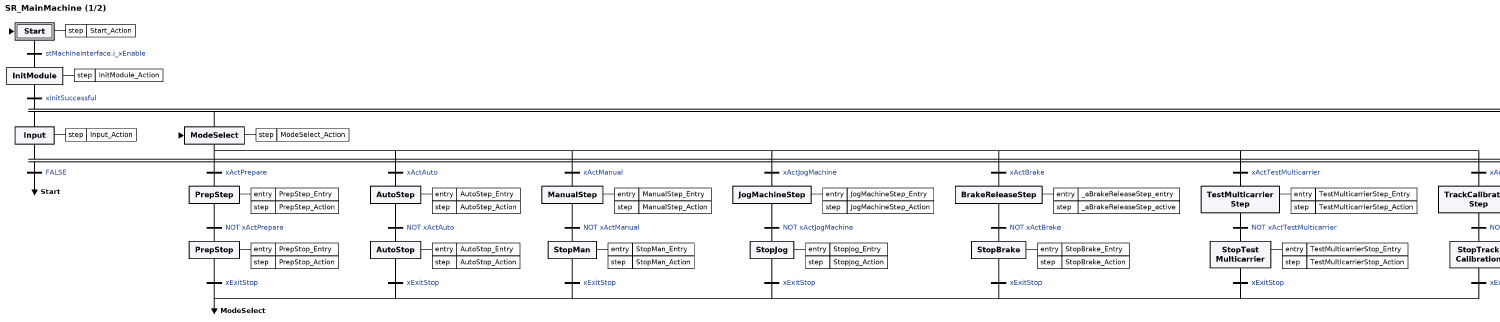
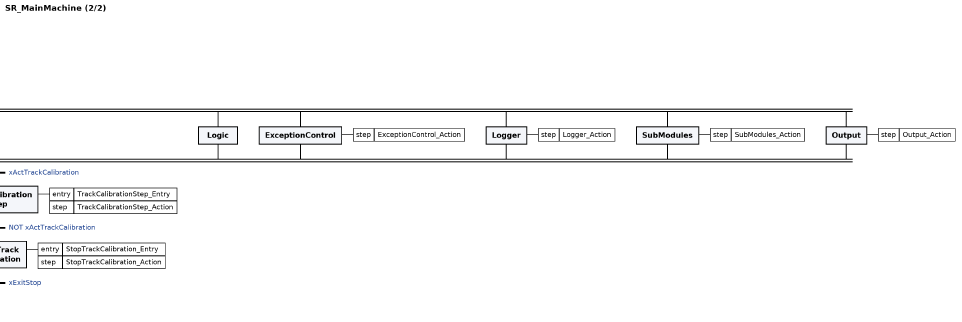
INITIAL_STEP Start:
    Start_Action(N);  // step action
END_STEP
TRANSITION FROM Start TO InitModule
    := stMachineInterface.i_xEnable;
END_TRANSITION
STEP InitModule:
    InitModule_Action(N);  // step action
END_STEP
TRANSITION FROM InitModule TO (Input, ModeSelect, Logic, ExceptionControl, Logger, SubModules, Output)
    := xInitSuccessful;
END_TRANSITION
STEP Input:
    Input_Action(N);  // step action
END_STEP
STEP ModeSelect:
    ModeSelect_Action(N);  // step action
END_STEP
TRANSITION FROM ModeSelect TO PrepStep
    := xActPrepare;
END_TRANSITION
STEP PrepStep:
    PrepStep_Entry(P1);  // entry action
    PrepStep_Action(N);  // step action
END_STEP
TRANSITION FROM PrepStep TO PrepStop
    := NOT xActPrepare;
END_TRANSITION
STEP PrepStop:
    PrepStop_Entry(P1);  // entry action
    PrepStop_Action(N);  // step action
END_STEP
TRANSITION FROM PrepStop TO ModeSelect
    := xExitStop;
END_TRANSITION
TRANSITION FROM ModeSelect TO AutoStep
    := xActAuto;
END_TRANSITION
STEP AutoStep:
    AutoStep_Entry(P1);  // entry action
    AutoStep_Action(N);  // step action
END_STEP
TRANSITION FROM AutoStep TO AutoStop
    := NOT xActAuto;
END_TRANSITION
STEP AutoStop:
    AutoStop_Entry(P1);  // entry action
    AutoStop_Action(N);  // step action
END_STEP
TRANSITION FROM AutoStop TO ModeSelect
    := xExitStop;
END_TRANSITION
TRANSITION FROM ModeSelect TO ManualStep
    := xActManual;
END_TRANSITION
STEP ManualStep:
    ManualStep_Entry(P1);  // entry action
    ManualStep_Action(N);  // step action
END_STEP
TRANSITION FROM ManualStep TO StopMan
    := NOT xActManual;
END_TRANSITION
STEP StopMan:
    StopMan_Entry(P1);  // entry action
    StopMan_Action(N);  // step action
END_STEP
TRANSITION FROM StopMan TO ModeSelect
    := xExitStop;
END_TRANSITION
TRANSITION FROM ModeSelect TO JogMachineStep
    := xActJogMachine;
END_TRANSITION
STEP JogMachineStep:
    JogMachineStep_Entry(P1);  // entry action
    JogMachineStep_Action(N);  // step action
END_STEP
TRANSITION FROM JogMachineStep TO StopJog
    := NOT xActJogMachine;
END_TRANSITION
STEP StopJog:
    StopJog_Entry(P1);  // entry action
    StopJog_Action(N);  // step action
END_STEP
TRANSITION FROM StopJog TO ModeSelect
    := xExitStop;
END_TRANSITION
TRANSITION FROM ModeSelect TO BrakeReleaseStep
    := xActBrake;
END_TRANSITION
STEP BrakeReleaseStep:
    _aBrakeReleaseStep_entry(P1);  // entry action
    _aBrakeReleaseStep_active(N);  // step action
END_STEP
TRANSITION FROM BrakeReleaseStep TO StopBrake
    := NOT xActBrake;
END_TRANSITION
STEP StopBrake:
    StopBrake_Entry(P1);  // entry action
    StopBrake_Action(N);  // step action
END_STEP
TRANSITION FROM StopBrake TO ModeSelect
    := xExitStop;
END_TRANSITION
TRANSITION FROM ModeSelect TO TestMulticarrierStep
    := xActTestMulticarrier;
END_TRANSITION
STEP TestMulticarrierStep:
    TestMulticarrierStep_Entry(P1);  // entry action
    TestMulticarrierStep_Action(N);  // step action
END_STEP
TRANSITION FROM TestMulticarrierStep TO StopTestMulticarrier
    := NOT xActTestMulticarrier;
END_TRANSITION
STEP StopTestMulticarrier:
    TestMulticarrierStop_Entry(P1);  // entry action
    TestMulticarrierStop_Action(N);  // step action
END_STEP
TRANSITION FROM StopTestMulticarrier TO ModeSelect
    := xExitStop;
END_TRANSITION
TRANSITION FROM ModeSelect TO TrackCalibrationStep
    := xActTrackCalibration;
END_TRANSITION
STEP TrackCalibrationStep:
    TrackCalibrationStep_Entry(P1);  // entry action
    TrackCalibrationStep_Action(N);  // step action
END_STEP
TRANSITION FROM TrackCalibrationStep TO StopTrackCalibration
    := NOT xActTrackCalibration;
END_TRANSITION
STEP StopTrackCalibration:
    StopTrackCalibration_Entry(P1);  // entry action
    StopTrackCalibration_Action(N);  // step action
END_STEP
TRANSITION FROM StopTrackCalibration TO ModeSelect
    := xExitStop;
END_TRANSITION
STEP Logic:
END_STEP
STEP ExceptionControl:
    ExceptionControl_Action(N);  // step action
END_STEP
STEP Logger:
    Logger_Action(N);  // step action
END_STEP
STEP SubModules:
    SubModules_Action(N);  // step action
END_STEP
STEP Output:
    Output_Action(N);  // step action
END_STEP
TRANSITION FROM (Input, Logic, ExceptionControl, Logger, SubModules, Output) TO Start
    := FALSE;
END_TRANSITION

ACTION Init_CmdTables:
(* System generated code, could be modified for your application *)

//-------------------------------------------------------------------------------------------------------------------
//-- Prepare  --
	//
	TPL.FC_FirstStep(udiStepIndex, diStep);
	astPrepareTable[udiStepIndex].sTitle					:= 'Prepare AllSubModules';
	astPrepareTable[udiStepIndex].udiModuleName				:= TPL.Gc_udiAllSubModules;
	astPrepareTable[udiStepIndex].diStep					:= diStep;
	astPrepareTable[udiStepIndex].diCMD						:= ET_Cmd.Prepare;
	astPrepareTable[udiStepIndex].timTimeOut				:= T#0MS;
	astPrepareTable[udiStepIndex].xEndCMD					:= FALSE;
	
	TPL.FC_LastStep(udiStepIndex, diStep);
	astPrepareTable[udiStepIndex].sTitle					:= 'End';
	astPrepareTable[udiStepIndex].udiModuleName				:= 0;
	astPrepareTable[udiStepIndex].diStep					:= diStep;
	astPrepareTable[udiStepIndex].diCMD						:= 0;
	astPrepareTable[udiStepIndex].timTimeOut				:= T#0MS;
	astPrepareTable[udiStepIndex].xEndCMD					:= TRUE;
	
	TPL.FC_FirstCmdTable(iq_udiTableIndex:= udiTableIndex);
	astListofCMDTables[udiTableIndex].diCMD					:= ET_Cmd.Prepare;
	astListofCMDTables[udiTableIndex].sTitle				:= 'Prepare';
	astListofCMDTables[udiTableIndex].udiNumberOfCmdSteps	:= udiStepIndex;

//-------------------------------------------------------------------------------------------------------------------
//-- StopPrepare  --
	//
	TPL.FC_FirstStep(udiStepIndex, diStep);
	astStopPrepareTable[udiStepIndex].sTitle					:= 'Stop Alpha + Bravo';
	astStopPrepareTable[udiStepIndex].udiModuleName				:= c_udiServoDrivesGroup;
	astStopPrepareTable[udiStepIndex].diStep					:= diStep;
	astStopPrepareTable[udiStepIndex].diCMD						:= ET_Cmd.Stop;
	astStopPrepareTable[udiStepIndex].timTimeOut				:= T#0MS;
	astStopPrepareTable[udiStepIndex].xEndCMD					:= FALSE;
	
	TPL.FC_NextStep(udiStepIndex, diStep);
	astStopPrepareTable[udiStepIndex].sTitle					:= 'Hold MultiCarrier';
	astStopPrepareTable[udiStepIndex].udiModuleName				:= c_udiMultiCarrier;
	astStopPrepareTable[udiStepIndex].diStep					:= diStep;
	astStopPrepareTable[udiStepIndex].diCMD						:= ET_Cmd.Hold;
	astStopPrepareTable[udiStepIndex].timTimeOut				:= T#0MS;
	astStopPrepareTable[udiStepIndex].xEndCMD					:= FALSE;
	
	TPL.FC_LastStep(udiStepIndex, diStep);
	astStopPrepareTable[udiStepIndex].sTitle					:= 'End';
	astStopPrepareTable[udiStepIndex].udiModuleName				:= 0;
	astStopPrepareTable[udiStepIndex].diStep					:= diStep;
	astStopPrepareTable[udiStepIndex].diCMD						:= 0;
	astStopPrepareTable[udiStepIndex].timTimeOut				:= T#0MS;
	astStopPrepareTable[udiStepIndex].xEndCMD					:= TRUE;
	
	TPL.FC_NextCmdTable(iq_udiTableIndex:= udiTableIndex);
	astListofCMDTables[udiTableIndex].diCMD						:= ET_Cmd.StopPrepare;
	astListofCMDTables[udiTableIndex].sTitle					:= 'StopPrepare';
	astListofCMDTables[udiTableIndex].udiNumberOfCmdSteps		:= udiStepIndex;
	
	
//-------------------------------------------------------------------------------------------------------------------
//-- Auto  --
	//
	TPL.FC_FirstStep(udiStepIndex, diStep);
	astAutoTable[udiStepIndex].sTitle						:= 'Auto Bravo';
	astAutoTable[udiStepIndex].udiModuleName				:= c_udiBravo;
	astAutoTable[udiStepIndex].diStep						:= diStep;
	astAutoTable[udiStepIndex].diCMD						:= ET_Cmd.Auto;
	astAutoTable[udiStepIndex].timTimeOut					:= T#0MS;
	astAutoTable[udiStepIndex].xEndCMD						:= FALSE;
	
	TPL.FC_NextStep(udiStepIndex, diStep);
	astAutoTable[udiStepIndex].sTitle						:= 'Auto Alpha';
	astAutoTable[udiStepIndex].udiModuleName				:= c_udiAlpha;
	astAutoTable[udiStepIndex].diStep						:= diStep;
	astAutoTable[udiStepIndex].diCMD						:= ET_Cmd.Auto;
	astAutoTable[udiStepIndex].timTimeOut					:= T#0MS;
	astAutoTable[udiStepIndex].xEndCMD						:= FALSE;
	
	TPL.FC_NextStep(udiStepIndex, diStep);
	astAutoTable[udiStepIndex].sTitle						:= 'Auto MultiCarrier';
	astAutoTable[udiStepIndex].udiModuleName				:= c_udiMultiCarrier;
	astAutoTable[udiStepIndex].diStep						:= diStep;
	astAutoTable[udiStepIndex].diCMD						:= ET_Cmd.Auto;
	astAutoTable[udiStepIndex].timTimeOut					:= T#0MS;
	astAutoTable[udiStepIndex].xEndCMD						:= FALSE;
	
	TPL.FC_LastStep(udiStepIndex, diStep);
	astAutoTable[udiStepIndex].sTitle						:= 'End';
	astAutoTable[udiStepIndex].udiModuleName				:= 0;
	astAutoTable[udiStepIndex].diStep						:= diStep;
	astAutoTable[udiStepIndex].diCMD						:= 0;
	astAutoTable[udiStepIndex].timTimeOut					:= T#0MS;
	astAutoTable[udiStepIndex].xEndCMD						:= TRUE;
	
	TPL.FC_NextCmdTable(iq_udiTableIndex:= udiTableIndex);
	astListofCMDTables[udiTableIndex].diCMD					:= ET_Cmd.Auto;
	astListofCMDTables[udiTableIndex].sTitle				:= 'Auto';
	astListofCMDTables[udiTableIndex].udiNumberOfCmdSteps	:= udiStepIndex;

//-------------------------------------------------------------------------------------------------------------------
//-- StopAuto --
	//
	TPL.FC_FirstStep(udiStepIndex, diStep);
	astStopAutoTable[udiStepIndex].sTitle					:= 'Hold Alpha';
	astStopAutoTable[udiStepIndex].udiModuleName			:= c_udiAlpha;
	astStopAutoTable[udiStepIndex].diStep					:= diStep;
	astStopAutoTable[udiStepIndex].diCMD					:= ET_Cmd.Hold;
	astStopAutoTable[udiStepIndex].timTimeOut				:= T#0MS;
	astStopAutoTable[udiStepIndex].xEndCMD					:= FALSE;
	
	TPL.FC_NextStep(udiStepIndex, diStep);
	astStopAutoTable[udiStepIndex].sTitle					:= 'Stop MultiCarrier';
	astStopAutoTable[udiStepIndex].udiModuleName			:= c_udiMultiCarrier;
	astStopAutoTable[udiStepIndex].diStep					:= diStep;
	astStopAutoTable[udiStepIndex].diCMD					:= ET_Cmd.Stop;
	astStopAutoTable[udiStepIndex].timTimeOut				:= T#0MS;
	astStopAutoTable[udiStepIndex].xEndCMD					:= FALSE;
	
	TPL.FC_LastStep(udiStepIndex, diStep);
	astStopAutoTable[udiStepIndex].sTitle					:= 'End';
	astStopAutoTable[udiStepIndex].udiModuleName			:= 0;
	astStopAutoTable[udiStepIndex].diStep					:= diStep;
	astStopAutoTable[udiStepIndex].diCMD					:= 0;
	astStopAutoTable[udiStepIndex].timTimeOut				:= T#0MS;
	astStopAutoTable[udiStepIndex].xEndCMD					:= TRUE;
	
	TPL.FC_NextCmdTable(iq_udiTableIndex:= udiTableIndex);
	astListofCMDTables[udiTableIndex].diCMD						:= ET_Cmd.StopAuto;
	astListofCMDTables[udiTableIndex].sTitle					:= 'StopAuto';
	astListofCMDTables[udiTableIndex].udiNumberOfCmdSteps		:= udiStepIndex;
	
	
	
//-------------------------------------------------------------------------------------------------------------------
//-- Manual  --
	//
	TPL.FC_FirstStep(udiStepIndex, diStep);
	astManualTable[udiStepIndex].sTitle						:= 'Stop AllSubModules';
	astManualTable[udiStepIndex].udiModuleName				:= TPL.Gc_udiAllSubModules;
	astManualTable[udiStepIndex].diStep						:= diStep;
	astManualTable[udiStepIndex].diCMD						:= ET_Cmd.Stop;
	astManualTable[udiStepIndex].timTimeOut					:= T#0MS;
	astManualTable[udiStepIndex].xEndCMD					:= FALSE;
	
	TPL.FC_NextStep(udiStepIndex, diStep);
	astManualTable[udiStepIndex].sTitle						:= 'Manual SlaveGroup';
	astManualTable[udiStepIndex].udiModuleName				:= TPL.Gc_udiAllSubModules;
	astManualTable[udiStepIndex].diStep						:= diStep;
	astManualTable[udiStepIndex].diCMD						:= ET_Cmd.Manual;
	astManualTable[udiStepIndex].timTimeOut					:= T#0MS;
	astManualTable[udiStepIndex].xEndCMD					:= FALSE;
	
	TPL.FC_LastStep(udiStepIndex, diStep);
	astManualTable[udiStepIndex].sTitle						:= 'End';
	astManualTable[udiStepIndex].udiModuleName				:= 0;
	astManualTable[udiStepIndex].diStep						:= diStep;
	astManualTable[udiStepIndex].diCMD						:= 0;
	astManualTable[udiStepIndex].timTimeOut					:= T#0MS;
	astManualTable[udiStepIndex].xEndCMD					:= TRUE;
	
	TPL.FC_NextCmdTable(iq_udiTableIndex:= udiTableIndex);
	astListofCMDTables[udiTableIndex].diCMD					:= ET_Cmd.Manual;
	astListofCMDTables[udiTableIndex].sTitle				:= 'Manual';
	astListofCMDTables[udiTableIndex].udiNumberOfCmdSteps	:= udiStepIndex;

//-------------------------------------------------------------------------------------------------------------------
//-- TestMulticarrier --
	//
	TPL.FC_FirstStep(udiStepIndex, diStep);
	astTestMulticarrierTable[udiStepIndex].sTitle						:= 'TestMulticarrier';
	astTestMulticarrierTable[udiStepIndex].udiModuleName				:= c_udiMultiCarrier;
	astTestMulticarrierTable[udiStepIndex].diStep						:= diStep;
	astTestMulticarrierTable[udiStepIndex].diCMD						:= ET_Cmd.TestMulticarrier;
	astTestMulticarrierTable[udiStepIndex].timTimeOut					:= T#0MS;
	astTestMulticarrierTable[udiStepIndex].xEndCMD						:= FALSE;
	
	TPL.FC_LastStep(udiStepIndex, diStep);
	astTestMulticarrierTable[udiStepIndex].sTitle						:= 'End';
	astTestMulticarrierTable[udiStepIndex].udiModuleName				:= 0;
	astTestMulticarrierTable[udiStepIndex].diStep						:= diStep;
	astTestMulticarrierTable[udiStepIndex].diCMD						:= 0;
	astTestMulticarrierTable[udiStepIndex].timTimeOut					:= T#0MS;
	astTestMulticarrierTable[udiStepIndex].xEndCMD						:= TRUE;
	
	TPL.FC_NextCmdTable(iq_udiTableIndex:= udiTableIndex);
	astListofCMDTables[udiTableIndex].diCMD					:= ET_Cmd.TestMulticarrier;
	astListofCMDTables[udiTableIndex].sTitle				:= 'TestMulticarrier';
	astListofCMDTables[udiTableIndex].udiNumberOfCmdSteps	:= udiStepIndex;
	
//-------------------------------------------------------------------------------------------------------------------
//-- TrackCalibration --
	//
	TPL.FC_FirstStep(udiStepIndex, diStep);
	astTrackCalibrationTable[udiStepIndex].sTitle						:= 'TrackCalibration';
	astTrackCalibrationTable[udiStepIndex].udiModuleName				:= c_udiMultiCarrier;
	astTrackCalibrationTable[udiStepIndex].diStep						:= diStep;
	astTrackCalibrationTable[udiStepIndex].diCMD						:= ET_Cmd.TrackCalibration;
	astTrackCalibrationTable[udiStepIndex].timTimeOut					:= T#0MS;
	astTrackCalibrationTable[udiStepIndex].xEndCMD						:= FALSE;
	
	TPL.FC_LastStep(udiStepIndex, diStep);
	astTrackCalibrationTable[udiStepIndex].sTitle						:= 'End';
	astTrackCalibrationTable[udiStepIndex].udiModuleName				:= 0;
	astTrackCalibrationTable[udiStepIndex].diStep						:= diStep;
	astTrackCalibrationTable[udiStepIndex].diCMD						:= 0;
	astTrackCalibrationTable[udiStepIndex].timTimeOut					:= T#0MS;
	astTrackCalibrationTable[udiStepIndex].xEndCMD						:= TRUE;
	
	TPL.FC_NextCmdTable(iq_udiTableIndex:= udiTableIndex);
	astListofCMDTables[udiTableIndex].diCMD					:= ET_Cmd.TrackCalibration;
	astListofCMDTables[udiTableIndex].sTitle				:= 'TrackCalibration';
	astListofCMDTables[udiTableIndex].udiNumberOfCmdSteps	:= udiStepIndex;
	
//-------------------------------------------------------------------------------------------------------------------
//-- Stop --
	//
	TPL.FC_FirstStep(udiStepIndex, diStep);
	astStopTable[udiStepIndex].sTitle						:= 'Stop AllSubModules';
	astStopTable[udiStepIndex].udiModuleName				:= TPL.Gc_udiAllSubModules;
	astStopTable[udiStepIndex].diStep						:= diStep;
	astStopTable[udiStepIndex].diCMD						:= ET_Cmd.Stop;
	astStopTable[udiStepIndex].timTimeOut					:= T#0MS;
	astStopTable[udiStepIndex].xEndCMD						:= FALSE;
	
	TPL.FC_LastStep(udiStepIndex, diStep);
	astStopTable[udiStepIndex].sTitle						:= 'End';
	astStopTable[udiStepIndex].udiModuleName				:= 0;
	astStopTable[udiStepIndex].diStep						:= diStep;
	astStopTable[udiStepIndex].diCMD						:= 0;
	astStopTable[udiStepIndex].timTimeOut					:= T#0MS;
	astStopTable[udiStepIndex].xEndCMD						:= TRUE;
	
	TPL.FC_NextCmdTable(iq_udiTableIndex:= udiTableIndex);
	astListofCMDTables[udiTableIndex].diCMD					:= ET_Cmd.Stop;
	astListofCMDTables[udiTableIndex].sTitle				:= 'Stop';
	astListofCMDTables[udiTableIndex].udiNumberOfCmdSteps	:= udiStepIndex;

//-------------------------------------------------------------------------------------------------------------------
//-- Start --
	//
	TPL.FC_FirstStep(udiStepIndex, diStep);
	astStartTable[udiStepIndex].sTitle						:= 'Start AllSubModules';
	astStartTable[udiStepIndex].udiModuleName				:= TPL.Gc_udiAllSubModules;
	astStartTable[udiStepIndex].diStep						:= diStep;
	astStartTable[udiStepIndex].diCMD						:= ET_Cmd.Start;
	astStartTable[udiStepIndex].timTimeOut					:= T#0MS;
	astStartTable[udiStepIndex].xEndCMD						:= FALSE;
	
	TPL.FC_LastStep(udiStepIndex, diStep);
	astStartTable[udiStepIndex].sTitle						:= 'End';
	astStartTable[udiStepIndex].udiModuleName				:= 0;
	astStartTable[udiStepIndex].diStep						:= diStep;
	astStartTable[udiStepIndex].diCMD						:= 0;
	astStartTable[udiStepIndex].timTimeOut					:= T#0MS;
	astStartTable[udiStepIndex].xEndCMD						:= TRUE;
	
	TPL.FC_NextCmdTable(iq_udiTableIndex:= udiTableIndex);
	astListofCMDTables[udiTableIndex].diCMD					:= ET_Cmd.Start;
	astListofCMDTables[udiTableIndex].sTitle				:= 'Start';
	astListofCMDTables[udiTableIndex].udiNumberOfCmdSteps	:= udiStepIndex;
	
//-------------------------------------------------------------------------------------------------------------------
//-- Abort --
	//
	TPL.FC_FirstStep(udiStepIndex, diStep);
	astAbortTable[udiStepIndex].sTitle						:= 'Abort AllSubModules';
	astAbortTable[udiStepIndex].udiModuleName				:= TPL.Gc_udiAllSubModules;
	astAbortTable[udiStepIndex].diStep						:= diStep;
	astAbortTable[udiStepIndex].diCMD						:= ET_Cmd.Abort;
	astAbortTable[udiStepIndex].timTimeOut					:= T#0MS;
	astAbortTable[udiStepIndex].xEndCMD						:= FALSE;
	
	TPL.FC_LastStep(udiStepIndex, diStep);
	astAbortTable[udiStepIndex].sTitle						:= 'End';
	astAbortTable[udiStepIndex].udiModuleName				:= 0;
	astAbortTable[udiStepIndex].diStep						:= diStep;
	astAbortTable[udiStepIndex].diCMD						:= 0;
	astAbortTable[udiStepIndex].timTimeOut					:= T#0MS;
	astAbortTable[udiStepIndex].xEndCMD						:= TRUE;
	
	TPL.FC_NextCmdTable(iq_udiTableIndex:= udiTableIndex);
	astListofCMDTables[udiTableIndex].diCMD					:= ET_Cmd.Abort;
	astListofCMDTables[udiTableIndex].sTitle				:= 'Abort';
	astListofCMDTables[udiTableIndex].udiNumberOfCmdSteps	:= udiStepIndex;

//-------------------------------------------------------------------------------------------------------------------
//-- Hold --
	//
	TPL.FC_FirstStep(udiStepIndex, diStep);
	astHoldTable[udiStepIndex].sTitle						:= 'Hold Alpha';
	astHoldTable[udiStepIndex].udiModuleName				:= c_udiAlpha;
	astHoldTable[udiStepIndex].diStep						:= diStep;
	astHoldTable[udiStepIndex].diCMD						:= ET_Cmd.Hold;
	astHoldTable[udiStepIndex].timTimeOut					:= T#0MS;
	astHoldTable[udiStepIndex].xEndCMD						:= FALSE;
	
	TPL.FC_LastStep(udiStepIndex, diStep);
	astHoldTable[udiStepIndex].sTitle						:= 'End';
	astHoldTable[udiStepIndex].udiModuleName				:= 0;
	astHoldTable[udiStepIndex].diStep						:= diStep;
	astHoldTable[udiStepIndex].diCMD						:= 0;
	astHoldTable[udiStepIndex].timTimeOut					:= T#0MS;
	astHoldTable[udiStepIndex].xEndCMD						:= TRUE;
	
	TPL.FC_NextCmdTable(iq_udiTableIndex:= udiTableIndex);
	astListofCMDTables[udiTableIndex].diCMD					:= ET_Cmd.Hold;
	astListofCMDTables[udiTableIndex].sTitle				:= 'Hold';
	astListofCMDTables[udiTableIndex].udiNumberOfCmdSteps	:= udiStepIndex;

//-------------------------------------------------------------------------------------------------------------------
//-- Hold for JogMachine --
	//
	TPL.FC_FirstStep(udiStepIndex, diStep);
	astHoldJogMachineTable[udiStepIndex].sTitle				:= 'Stop Alpha';
	astHoldJogMachineTable[udiStepIndex].udiModuleName		:= c_udiAlpha;
	astHoldJogMachineTable[udiStepIndex].diStep				:= diStep;
	astHoldJogMachineTable[udiStepIndex].diCMD				:= ET_Cmd.Stop;
	astHoldJogMachineTable[udiStepIndex].timTimeOut			:= T#0MS;
	astHoldJogMachineTable[udiStepIndex].xEndCMD			:= FALSE;
	
	TPL.FC_LastStep(udiStepIndex, diStep);
	astHoldJogMachineTable[udiStepIndex].sTitle				:= 'End';
	astHoldJogMachineTable[udiStepIndex].udiModuleName		:= 0;
	astHoldJogMachineTable[udiStepIndex].diStep				:= diStep;
	astHoldJogMachineTable[udiStepIndex].diCMD				:= 0;
	astHoldJogMachineTable[udiStepIndex].timTimeOut			:= T#0MS;
	astHoldJogMachineTable[udiStepIndex].xEndCMD			:= TRUE;
	
	TPL.FC_NextCmdTable(iq_udiTableIndex:= udiTableIndex);
	astListofCMDTables[udiTableIndex].diCMD					:= ET_Cmd.HoldJM;
	astListofCMDTables[udiTableIndex].sTitle				:= 'Hold Jog Machine';
	astListofCMDTables[udiTableIndex].udiNumberOfCmdSteps	:= udiStepIndex;
//-------------------------------------------------------------------------------------------------------------------
//-- Brake Release --
	//
	TPL.FC_FirstStep(udiStepIndex, diStep);
	astBrakeReleaseTable[udiStepIndex].sTitle				:= 'BrakeRelease Bravo';
	astBrakeReleaseTable[udiStepIndex].udiModuleName		:= c_udiBravo;
	astBrakeReleaseTable[udiStepIndex].diStep				:= diStep;
	astBrakeReleaseTable[udiStepIndex].diCMD				:= ET_Cmd.BrakeRelease;
	astBrakeReleaseTable[udiStepIndex].timTimeOut			:= T#0MS;
	astBrakeReleaseTable[udiStepIndex].xEndCMD				:= FALSE;
	
	TPL.FC_LastStep(udiStepIndex, diStep);
	astBrakeReleaseTable[udiStepIndex].sTitle				:= 'End';
	astBrakeReleaseTable[udiStepIndex].udiModuleName		:= 0;
	astBrakeReleaseTable[udiStepIndex].diStep				:= diStep;
	astBrakeReleaseTable[udiStepIndex].diCMD				:= 0;
	astBrakeReleaseTable[udiStepIndex].timTimeOut			:= T#0MS;
	astBrakeReleaseTable[udiStepIndex].xEndCMD				:= TRUE;
	
	TPL.FC_NextCmdTable(iq_udiTableIndex:= udiTableIndex);
	astListofCMDTables[udiTableIndex].diCMD					:= ET_Cmd.BrakeRelease;
	astListofCMDTables[udiTableIndex].sTitle				:= 'BrakeRelease';
	astListofCMDTables[udiTableIndex].udiNumberOfCmdSteps	:= udiStepIndex;

//-------------------------------------------------------------------------------------------------------------------
//-- JogMachine --
	//
	TPL.FC_FirstStep(udiStepIndex, diStep);
	astJogMachineTable[udiStepIndex].sTitle					:= 'Auto Bravo';
	astJogMachineTable[udiStepIndex].udiModuleName			:= c_udiBravo;
	astJogMachineTable[udiStepIndex].diStep					:= diStep;
	astJogMachineTable[udiStepIndex].diCMD					:= ET_Cmd.Auto;
	astJogMachineTable[udiStepIndex].timTimeOut				:= T#0MS;
	astJogMachineTable[udiStepIndex].xEndCMD				:= FALSE;
	TPL.FC_NextStep(udiStepIndex, diStep);
	astJogMachineTable[udiStepIndex].sTitle					:= 'Manual Alpha';
	astJogMachineTable[udiStepIndex].udiModuleName			:= c_udiAlpha;
	astJogMachineTable[udiStepIndex].diStep					:= diStep;
	astJogMachineTable[udiStepIndex].diCMD					:= ET_Cmd.Manual;
	astJogMachineTable[udiStepIndex].timTimeOut				:= T#0MS;
	astJogMachineTable[udiStepIndex].xEndCMD				:= FALSE;
	
	TPL.FC_LastStep(udiStepIndex, diStep);
	astJogMachineTable[udiStepIndex].sTitle					:= 'End';
	astJogMachineTable[udiStepIndex].udiModuleName			:= 0;
	astJogMachineTable[udiStepIndex].diStep					:= diStep;
	astJogMachineTable[udiStepIndex].diCMD					:= 0;
	astJogMachineTable[udiStepIndex].timTimeOut				:= T#0MS;
	astJogMachineTable[udiStepIndex].xEndCMD				:= TRUE;
	
	TPL.FC_NextCmdTable(iq_udiTableIndex:= udiTableIndex);
	astListofCMDTables[udiTableIndex].diCMD					:= ET_Cmd.Jogging;
	astListofCMDTables[udiTableIndex].sTitle				:= 'Jogging';
	astListofCMDTables[udiTableIndex].udiNumberOfCmdSteps	:= udiStepIndex;

	
//-------------------------------------------------------------------------------------------------------------------
(* End of system generated code, could be modified for your application *)
END_ACTION

ACTION Init_SubModules:
(* System generated code, could be modified for your application *)

(* Module Group declaration *)

aaudiSubModuleGroups[c_udiMasterGroup-TPL.Gc_udiGroupOffset,TPL.ET_Group.Member1]	:= c_udiAlpha;		(* The c_udiAlpha is the first element of the group c_udiMasterGroup *)
aaudiSubModuleGroups[c_udiMasterGroup-TPL.Gc_udiGroupOffset,TPL.ET_Group.Member2]	:= 0;				(* There is no second element of the group c_udiMasterGroup *)

aaudiSubModuleGroups[c_udiServoDrivesGroup-TPL.Gc_udiGroupOffset,TPL.ET_Group.Member1]	:= c_udiBravo;		(* The c_udiBravo is the first element of the group c_udiServoDrivesGroup *)
aaudiSubModuleGroups[c_udiServoDrivesGroup-TPL.Gc_udiGroupOffset,TPL.ET_Group.Member2]	:= c_udiAlpha;		(* The c_udiCharly is the second element of the group c_udiServoDrivesGroup *)


(* Configuration of exception logging *)
G_stLogDataList.wExceptionLogDataFilter	:= UDINT_TO_WORD(TPL.ET_LogDataFilter.ExceptionListDefault);

(* Exception in case of an overflow of the exception list - Set ModuleId and ModuleName *)
G_stExceptionList.stOverflowException.udiModuleId	:= stMachineInterface.i_udiModuleId;
G_stExceptionList.stOverflowException.sModuleName	:= stMachineInterface.i_sModuleName;


(* Example, how to modify the reaction of the overflow exception, by default all reactions are set *)
// FC_ReinitReaction(iq_stException := G_stExceptionList.stOverflowError); //set reaction to no reaction
// G_stExceptionList.stOverflowException.stReaction.axReaction[TPL.ET_Reaction.AsyncStop] := TRUE;
// G_stExceptionList.stOverflowException.stReaction.axReaction[TPL.ET_Reaction.MainsContactorOff] := TRUE; //ensure that the worst possible reactions for your machine are set


(* Set logger save file name and path *)
G_stLoggerInterface.i_sFileName		:= 'ram0:TPL_LOG.XML';					(* 'ide0:TPL_LOG.XML', 'ram0:TPL_LOG.CSV', 'remote:ram0:\\TPL_LOG.XML' *)
G_stLoggerInterface.i_xEnable		:= TRUE;
G_stLoggerInterface.i_etSortKey		:= TPL.ET_LogDataSortKey.SortByTime;	(*	TPL.ET_LogDataSortKey.SortByCmd
																				TPL.ET_LogDataSortKey.SortById
																				TPL.ET_LogDataSortKey.SortByModuleId
																				TPL.ET_LogDataSortKey.SortByModuleIdAndTime
																				TPL.ET_LogDataSortKey.SortByName
																				TPL.ET_LogDataSortKey.SortByReaction
																				TPL.ET_LogDataSortKey.SortByTime *)

(* End of system generated code, could be modified for your application *)

(* System generated code, do not change without consulting 'Schneider Electric Automation GmbH' - otherwise you risk instability!!!*)
xInitSubModulesException := FALSE;

(*****************************************************************************************************************************************************)
(* Set IDs of SubModules *)	

TPL.FC_SetSubModuleIds(	i_udiMainModuleID			:= stMachineInterface.i_udiModuleId,
						i_pstSubModulesItf			:= ADR(astSubModuleInterface),
						i_udiNumberOfSubModules		:= c_udiNumberOfSubModules,
						q_etDiag					=> etDiag,
						q_etDiagExt					=> etDiagExtTPL);
					
IF etDiag <> GD.ET_Diag.Ok AND NOT xInitSubModulesException THEN
	xInitSubModulesException := TRUE;
	
	stInitSubModulesException.sMsg := PDL.FC_MultiConcat(	i_sString1 := 'SetSubModuleIds - ', 
															i_sString2 := GD.FC_EtDiagToString(i_etDiag := etDiag), 
															i_sString3 := ' - ', 
															i_sString4 := TPL.FC_EtDiagExtToString(i_etDiagExt := etDiagExtTPL));
END_IF	

(*****************************************************************************************************************************************************)
(* Set exception if any exception occurred *)

fbExceptionHandler.SetException(i_xExceptionActive	:= xInitSubModulesException, 
								iq_stException		:= stInitSubModulesException, 
								iq_stExceptionList	:= G_stExceptionList);

xInitSuccessful := xInitSuccessful AND NOT xInitSubModulesException;
					
etDiag := GD.ET_Diag.Ok;
					
(* End of system generated code, do not change without consulting 'Schneider Electric Automation GmbH' - otherwise you risk instability!!!*)
END_ACTION

ACTION Init_Alpha:
(* System generated code, could be modified for your application *)

(* AlphaModule *)
astSubModuleInterface[c_udiAlpha].i_sModuleName		:= STANDARD.CONCAT(STR1 := stMachineInterface.i_sModuleName, STR2 := ': Alpha');
astSubModuleInterface[c_udiAlpha].i_xLogEnable		:= TRUE;
astSubModuleInterface[c_udiAlpha].i_wLogDataFilter	:= UDINT_TO_WORD(TPL.ET_LogDataFilter.ModuleDefault);

SR_AlphaModule.RegisterLoggerPoint(	i_ifParent	:= fbLoggerPoint,
									i_sName		:= 'Alpha',
									q_etDiag	=> ,
									q_etDiagExt	=> );
								

(* End of system generated code, could be modified for your application *)
END_ACTION

ACTION Init_Bravo:
(* System generated code, could be modified for your application *)

(* BravoModule *)
astSubModuleInterface[c_udiBravo].i_sModuleName		:= STANDARD.CONCAT(STR1 := stMachineInterface.i_sModuleName, STR2 := ': Bravo');
astSubModuleInterface[c_udiBravo].i_xLogEnable		:= TRUE;
astSubModuleInterface[c_udiBravo].i_wLogDataFilter	:= UDINT_TO_WORD(TPL.ET_LogDataFilter.ModuleDefault);

SR_BravoModule.RegisterLoggerPoint(	i_ifParent	:= fbLoggerPoint,
									i_sName		:= 'Bravo',
									q_etDiag	=> ,
									q_etDiagExt	=> );

(* End of system generated code, could be modified for your application *)
END_ACTION

ACTION Init_MultiCarrier:
(* System generated code, could be modified for your application *)

(* CharlyModule *)
astSubModuleInterface[c_udiMultiCarrier].i_sModuleName	:= STANDARD.CONCAT(STR1 := stMachineInterface.i_sModuleName, STR2 := ': MultiCarrier');
astSubModuleInterface[c_udiMultiCarrier].i_xLogEnable		:= TRUE;
astSubModuleInterface[c_udiMultiCarrier].i_wLogDataFilter	:= UDINT_TO_WORD(TPL.ET_LogDataFilter.ModuleDefault);

SR_MultiCarrierModule.RegisterLoggerPoint(	i_ifParent	:= fbLoggerPoint,
											i_sName		:= 'MultiCarrier',
											q_etDiag	=> ,
											q_etDiagExt	=> );

(* End of system generated code, could be modified for your application *)
END_ACTION

ACTION ExceptionControl_Action:
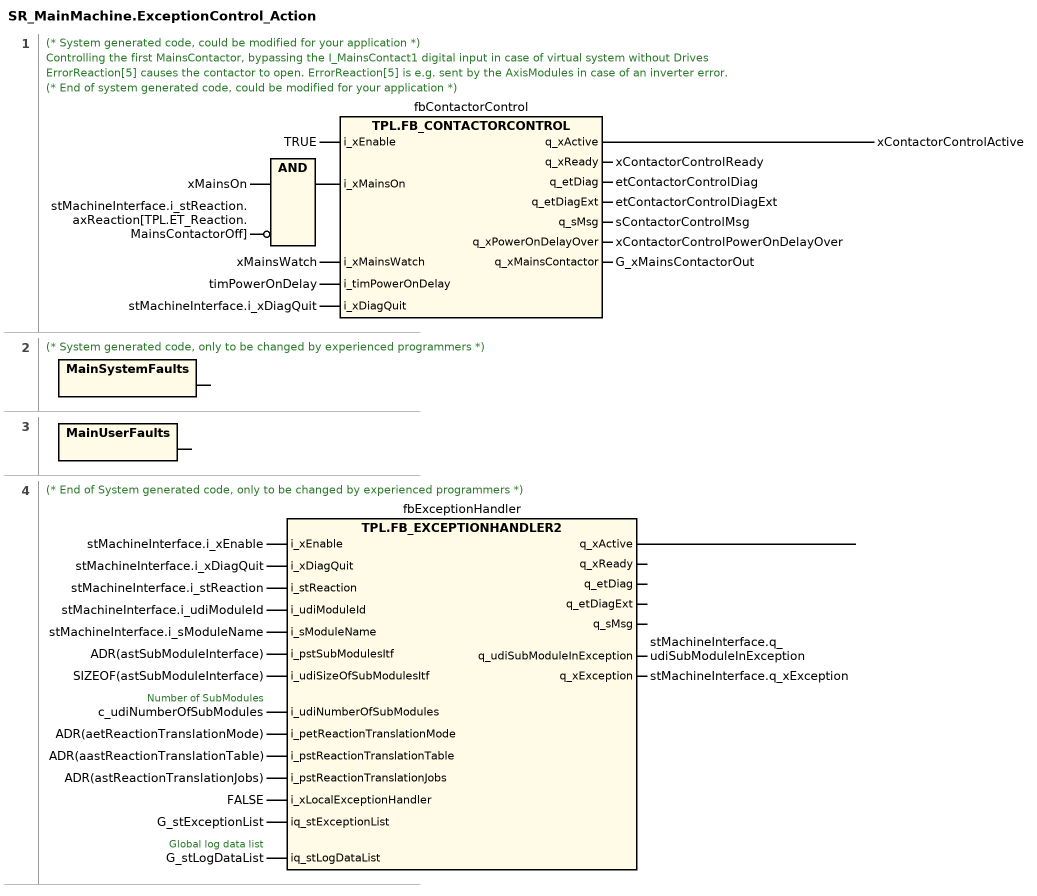
// NETWORK 1
// 					(* System generated code, could be modified for your application *)
// Controlling the first MainsContactor, bypassing the I_MainsContact1 digital input in case of virtual system without Drives
// ErrorReaction[5] causes the contactor to open. ErrorReaction[5] is e.g. sent by the AxisModules in case of an inverter error.
// (* End of system generated code, could be modified for your application *)
//
//   fbContactorControl: Contactor Control related variables
fbContactorControl(
    i_xEnable := TRUE,
    i_xMainsOn := xMainsOn AND NOT stMachineInterface.i_stReaction.axReaction[TPL.ET_Reaction.MainsContactorOff],
    i_xMainsWatch := xMainsWatch,
    i_timPowerOnDelay := timPowerOnDelay,
    i_xDiagQuit := stMachineInterface.i_xDiagQuit,
    q_xReady => xContactorControlReady,
    q_etDiag => etContactorControlDiag,
    q_etDiagExt => etContactorControlDiagExt,
    q_sMsg => sContactorControlMsg,
    q_xPowerOnDelayOver => xContactorControlPowerOnDelayOver,
    q_xMainsContactor => G_xMainsContactorOut); // TPL.FB_CONTACTORCONTROL
xContactorControlActive := fbContactorControl.q_xActive;

// NETWORK 2
// (* System generated code, only to be changed by experienced programmers *)
MainSystemFaults();

// NETWORK 3
MainUserFaults();

// NETWORK 4
// (* End of System generated code, only to be changed by experienced programmers *)
//   fbExceptionHandler: ExceptionHandling related variables
//   c_udiNumberOfSubModules: Number of SubModules
//   G_stLogDataList: Global log data list
fbExceptionHandler(
    i_xEnable := stMachineInterface.i_xEnable,
    i_xDiagQuit := stMachineInterface.i_xDiagQuit,
    i_stReaction := stMachineInterface.i_stReaction,
    i_udiModuleId := stMachineInterface.i_udiModuleId,
    i_sModuleName := stMachineInterface.i_sModuleName,
    i_pstSubModulesItf := ADR(astSubModuleInterface),
    i_udiSizeOfSubModulesItf := SIZEOF(astSubModuleInterface),
    i_udiNumberOfSubModules := c_udiNumberOfSubModules,
    i_petReactionTranslationMode := ADR(aetReactionTranslationMode),
    i_pstReactionTranslationTable := ADR(aastReactionTranslationTable),
    i_pstReactionTranslationJobs := ADR(astReactionTranslationJobs),
    i_xLocalExceptionHandler := FALSE,
    iq_stExceptionList := G_stExceptionList,
    iq_stLogDataList := G_stLogDataList,
    q_udiSubModuleInException => stMachineInterface.q_udiSubModuleInException,
    q_xException => stMachineInterface.q_xException); // TPL.FB_EXCEPTIONHANDLER2
END_ACTION

ACTION Init_Exceptions:
(* System generated code, could be modified for your application *)

(*
	TPL.ET_Reaction.AsyncStop
	TPL.ET_Reaction.SyncStopEL
	TPL.ET_Reaction.SyncStopEH
	TPL.ET_Reaction.StopEndOfCycle
	TPL.ET_Reaction.MainsContactorOff
*)

(*------------------------------------------------------------------------------------------*)
(* Init System Exceptions *)
(*------------------------------------------------------------------------------------------*)

stSystemException1.etDiag														:= GD.ET_Diag.Ok; (* Replaced on usage *)
stSystemException1.udiDiagExt													:= ET_DiagExt.Ok; (* Replaced on usage *)
stSystemException1.sDiagExt														:= FC_EtDiagExtToString(ET_DiagExt.Ok); (* Replaced on usage *)
stSystemException1.sMsg															:= ''; (* Replaced on usage *)
stSystemException1.udiModuleId													:= stMachineInterface.i_udiModuleId;
stSystemException1.sModuleName													:= stMachineInterface.i_sModuleName;
stSystemException1.etSource														:= TPL.ET_ExceptionSource.Main;
stSystemException1.timDelayTime													:= T#0MS;
stSystemException1.wHmiAttributes												:= 0;
stSystemException1.xAutoQuit													:= FALSE;
stSystemException1.stReaction.axReaction[TPL.ET_Reaction.AsyncStop]				:= TRUE;

stSystemException2.etDiag														:= GD.ET_Diag.Ok; (* Replaced on usage *)
stSystemException2.udiDiagExt													:= ET_DiagExt.Ok; (* Replaced on usage *)
stSystemException2.sDiagExt														:= FC_EtDiagExtToString(ET_DiagExt.Ok); (* Replaced on usage *)
stSystemException2.sMsg															:= ''; (* Replaced on usage *)
stSystemException2.udiModuleId													:= stMachineInterface.i_udiModuleId;
stSystemException2.sModuleName													:= stMachineInterface.i_sModuleName;
stSystemException2.etSource														:= TPL.ET_ExceptionSource.Main;
stSystemException2.timDelayTime													:= T#0MS;
stSystemException2.wHmiAttributes												:= 0;
stSystemException2.xAutoQuit													:= FALSE;
stSystemException2.stReaction.axReaction[TPL.ET_Reaction.SyncStopEL]			:= TRUE;

stSystemException3.etDiag														:= GD.ET_Diag.Ok; (* Replaced on usage *)
stSystemException3.udiDiagExt													:= ET_DiagExt.Ok; (* Replaced on usage *)
stSystemException3.sDiagExt														:= FC_EtDiagExtToString(ET_DiagExt.Ok); (* Replaced on usage *)
stSystemException3.sMsg															:= ''; (* Replaced on usage *)
stSystemException3.udiModuleId													:= stMachineInterface.i_udiModuleId;
stSystemException3.sModuleName													:= stMachineInterface.i_sModuleName;
stSystemException3.etSource														:= TPL.ET_ExceptionSource.Main;
stSystemException3.timDelayTime													:= T#0MS;
stSystemException3.wHmiAttributes												:= 0;
stSystemException3.xAutoQuit													:= FALSE;
stSystemException3.stReaction.axReaction[TPL.ET_Reaction.SyncStopEH]			:= TRUE;

stEmergencyStopException.etDiag													:= GD.ET_Diag.ExecutionAborted;
stEmergencyStopException.udiDiagExt												:= ET_DiagExt.MainSystemEmergencyStop;
stEmergencyStopException.sDiagExt												:= FC_EtDiagExtToString(ET_DiagExt.MainSystemEmergencyStop);
stEmergencyStopException.sMsg													:= 'Emergency Stop';
stEmergencyStopException.udiModuleId											:= stMachineInterface.i_udiModuleId;
stEmergencyStopException.sModuleName											:= stMachineInterface.i_sModuleName;
stEmergencyStopException.etSource												:= TPL.ET_ExceptionSource.Main;
stEmergencyStopException.timDelayTime											:= T#0MS;
stEmergencyStopException.wHmiAttributes											:= 0;
stEmergencyStopException.xAutoQuit												:= FALSE;
stEmergencyStopException.stReaction.axReaction[TPL.ET_Reaction.SyncStopEL]		:= TRUE;

stContactorControlException.etDiag												:= GD.ET_Diag.Ok; (* Replaced on usage *)
stContactorControlException.udiDiagExt											:= ET_DiagExt.Ok; (* Replaced on usage *)
stContactorControlException.sDiagExt											:= FC_EtDiagExtToString(ET_DiagExt.Ok); (* Replaced on usage *)
stContactorControlException.sMsg												:= ''; (* Replaced on usage *)
stContactorControlException.udiModuleId											:= stMachineInterface.i_udiModuleId;
stContactorControlException.sModuleName											:= stMachineInterface.i_sModuleName;
stContactorControlException.etSource											:= TPL.ET_ExceptionSource.Main;
stContactorControlException.timDelayTime										:= T#0MS;
stContactorControlException.wHmiAttributes										:= 0;
stContactorControlException.xAutoQuit											:= FALSE;
stContactorControlException.stReaction.axReaction[TPL.ET_Reaction.AsyncStop]	:= TRUE;

stUpdateStructsException.etDiag													:= GD.ET_Diag.UnexpectedProgramBehavior;
stUpdateStructsException.udiDiagExt												:= ET_DiagExt.UpdateStructsException;
stUpdateStructsException.sDiagExt												:= FC_EtDiagExtToString(stUpdateStructsException.udiDiagExt);
stUpdateStructsException.sMsg													:= '';	(* Replaced on usage *)
stUpdateStructsException.udiModuleId											:= stMachineInterface.i_udiModuleId;
stUpdateStructsException.sModuleName											:= stMachineInterface.i_sModuleName;
stUpdateStructsException.stReaction.axReaction[TPL.ET_Reaction.AsyncStop]		:= TRUE;
stUpdateStructsException.etSource												:= TPL.ET_ExceptionSource.Main;
stUpdateStructsException.timDelayTime											:= T#0MS;
stUpdateStructsException.wHmiAttributes											:= 0;
stUpdateStructsException.xAutoQuit												:= FALSE;

stInitReactionsException.etDiag													:= GD.ET_Diag.UnexpectedProgramBehavior;
stInitReactionsException.udiDiagExt												:= ET_DiagExt.InitReactionsException;
stInitReactionsException.sDiagExt												:= FC_EtDiagExtToString(stInitReactionsException.udiDiagExt);
stInitReactionsException.sMsg													:= '';	(* Replaced on usage *)
stInitReactionsException.udiModuleId											:= stMachineInterface.i_udiModuleId;
stInitReactionsException.sModuleName											:= stMachineInterface.i_sModuleName;
stInitReactionsException.stReaction.axReaction[TPL.ET_Reaction.AsyncStop]		:= TRUE;
stInitReactionsException.etSource												:= TPL.ET_ExceptionSource.Main;
stInitReactionsException.timDelayTime											:= T#0MS;
stInitReactionsException.wHmiAttributes											:= 0;
stInitReactionsException.xAutoQuit												:= FALSE;

stInitSubModulesException.etDiag												:= GD.ET_Diag.UnexpectedProgramBehavior;
stInitSubModulesException.udiDiagExt											:= ET_DiagExt.InitSubModulesException;
stInitSubModulesException.sDiagExt												:= FC_EtDiagExtToString(stInitSubModulesException.udiDiagExt);
stInitSubModulesException.sMsg													:= '';	(* Replaced on usage *)
stInitSubModulesException.udiModuleId											:= stMachineInterface.i_udiModuleId;
stInitSubModulesException.sModuleName											:= stMachineInterface.i_sModuleName;
stInitSubModulesException.stReaction.axReaction[TPL.ET_Reaction.AsyncStop]		:= TRUE;
stInitSubModulesException.etSource												:= TPL.ET_ExceptionSource.Main;
stInitSubModulesException.timDelayTime											:= T#0MS;
stInitSubModulesException.wHmiAttributes										:= 0;
stInitSubModulesException.xAutoQuit												:= FALSE;

(*------------------------------------------------------------------------------------------*)
(* Init User Exceptions *)
(*------------------------------------------------------------------------------------------*)	

stUserException1.etDiag															:= GD.ET_Diag.ExecutionAborted; (* Replaced on usage *)
stUserException1.udiDiagExt														:= ET_DiagExtUser.Exception1FromMain; (* Replaced on usage *)
stUserException1.sDiagExt														:= FC_EtDiagExtUserToString(stUserException1.udiDiagExt); (* Replaced on usage *)
//stUserException1.sMsg															:= 'User Exception 1'; (* To be replaced if used *)
stUserException1.udiModuleId													:= stMachineInterface.i_udiModuleId;
stUserException1.sModuleName													:= stMachineInterface.i_sModuleName;
stUserException1.etSource														:= TPL.ET_ExceptionSource.User;
stUserException1.timDelayTime													:= T#0MS;
stUserException1.wHmiAttributes													:= 0;
stUserException1.xAutoQuit														:= FALSE;
stUserException1.stReaction.axReaction[TPL.ET_Reaction.AsyncStop]				:= TRUE;

stUserException2.etDiag															:= GD.ET_Diag.ExecutionAborted; (* Replaced on usage *)
stUserException2.udiDiagExt														:= ET_DiagExtUser.Exception2FromMain; (* Replaced on usage *)
stUserException2.sDiagExt														:= FC_EtDiagExtUserToString(stUserException2.udiDiagExt); (* Replaced on usage *)
stUserException2.sMsg															:= 'User Exception 2'; (* To be replaced if used *)
stUserException2.udiModuleId													:= stMachineInterface.i_udiModuleId;
stUserException2.sModuleName													:= stMachineInterface.i_sModuleName;
stUserException2.etSource														:= TPL.ET_ExceptionSource.User;
stUserException2.timDelayTime													:= T#0MS;
stUserException2.wHmiAttributes													:= 0;
stUserException2.xAutoQuit														:= FALSE;
stUserException2.stReaction.axReaction[TPL.ET_Reaction.SyncStopEL]				:= TRUE;

stUserException3.etDiag															:= GD.ET_Diag.ExecutionAborted; (* Replaced on usage *)
stUserException3.udiDiagExt														:= ET_DiagExtUser.Exception3FromMain; (* Replaced on usage *)
stUserException3.sDiagExt														:= FC_EtDiagExtUserToString(stUserException3.udiDiagExt); (* Replaced on usage *)
stUserException3.sMsg															:= 'User Exception 3'; (* To be replaced if used *)
stUserException3.udiModuleId													:= stMachineInterface.i_udiModuleId;
stUserException3.sModuleName													:= stMachineInterface.i_sModuleName;
stUserException3.etSource														:= TPL.ET_ExceptionSource.User;
stUserException3.timDelayTime													:= T#0MS;
stUserException3.wHmiAttributes													:= 0;
stUserException3.xAutoQuit														:= TRUE;
stUserException3.stReaction.axReaction[TPL.ET_Reaction.SyncStopEH]				:= TRUE;

stUserException4.etDiag															:= GD.ET_Diag.ExecutionAborted; (* Replaced on usage *)
stUserException4.udiDiagExt														:= ET_DiagExtUser.Exception4FromMain; (* Replaced on usage *)
stUserException4.sDiagExt														:= FC_EtDiagExtUserToString(stUserException4.udiDiagExt); (* Replaced on usage *)
stUserException4.sMsg															:= 'User Exception 4'; (* To be replaced if used *)	
stUserException4.udiModuleId													:= stMachineInterface.i_udiModuleId;
stUserException4.sModuleName													:= stMachineInterface.i_sModuleName;
stUserException4.etSource														:= TPL.ET_ExceptionSource.User;
stUserException4.timDelayTime													:= T#0MS;
stUserException4.wHmiAttributes													:= 0;
stUserException4.xAutoQuit														:= FALSE;
stUserException4.stReaction.axReaction[TPL.ET_Reaction.StopEndOfCycle]			:= TRUE;

stUserException5.etDiag															:= GD.ET_Diag.ExecutionAborted; (* Replaced on usage *)
stUserException5.udiDiagExt														:= ET_DiagExtUser.Exception5FromMain; (* Replaced on usage *)
stUserException5.sDiagExt														:= FC_EtDiagExtUserToString(stUserException5.udiDiagExt); (* Replaced on usage *)
stUserException5.sMsg															:= 'User Exception 5'; (* To be replaced if used *)		
stUserException5.udiModuleId													:= stMachineInterface.i_udiModuleId;
stUserException5.sModuleName													:= stMachineInterface.i_sModuleName;
stUserException5.etSource														:= TPL.ET_ExceptionSource.User;
stUserException5.timDelayTime													:= T#0MS;
stUserException5.wHmiAttributes													:= 0;
stUserException5.xAutoQuit														:= FALSE;
stUserException5.stReaction.axReaction[TPL.ET_Reaction.MainsContactorOff]		:= TRUE;
stUserException5.stReaction.axReaction[TPL.ET_Reaction.StopEndOfCycle]			:= TRUE;

(* End of system generated code, could be modified for your application *)
END_ACTION

ACTION Init_Reactions:
(* System generated code, only to be changed by experienced programmers *)
IF c_udiNumberOfSubModules < 1 THEN
	RETURN;
END_IF

(* Change of default reactions only on demand *)

xInitReactionsException := FALSE;

(*****************************************************************************************************************************************************)
(* Init ReactionTranslationMode *)

TPL.FC_InitReactionTranslationMode(	i_udiNumberOfSubModules			:= c_udiNumberOfSubModules,
									i_petReactionTranslationMode	:= ADR(aetReactionTranslationMode),
									q_etDiag						=> etDiag,
									q_etDiagExt						=> etDiagExtTPL);
							
IF etDiag <> GD.ET_Diag.Ok AND NOT xInitReactionsException THEN
	xInitReactionsException := TRUE;
	
	stInitReactionsException.sMsg := PDL.FC_MultiConcat(i_sString1 := 'InitReactionTranslationMode - ', 
														i_sString2 := GD.FC_EtDiagToString(i_etDiag := etDiag), 
														i_sString3 := ' - ', 
														i_sString4 := TPL.FC_EtDiagExtToString(i_etDiagExt := etDiagExtTPL));
END_IF	

(*****************************************************************************************************************************************************)
(* Init ReactionTranslationTable *)	

TPL.FC_InitReactionTranslationTable(i_udiNumberOfSubModules			:= c_udiNumberOfSubModules,
									i_pstReactionTranslationTable	:= ADR(aastReactionTranslationTable),
									q_etDiag						=> etDiag,
									q_etDiagExt						=> etDiagExtTPL);
									
IF etDiag <> GD.ET_Diag.Ok AND NOT xInitReactionsException THEN
	xInitReactionsException := TRUE;
	
	stInitReactionsException.sMsg := PDL.FC_MultiConcat(i_sString1 := 'InitReactionTranslationTable - ', 
														i_sString2 := GD.FC_EtDiagToString(i_etDiag := etDiag), 
														i_sString3 := ' - ', 
														i_sString4 := TPL.FC_EtDiagExtToString(i_etDiagExt := etDiagExtTPL));
END_IF		

(*****************************************************************************************************************************************************)
(* Init ReactionTranslationJobs *)	
								
TPL.FC_InitReactionTranslationJobs( i_udiNumberOfSubModules			:= c_udiNumberOfSubModules,
									i_pstReactionTranslationJobs	:= ADR(astReactionTranslationJobs),
									q_etDiag						=> etDiag,
									q_etDiagExt						=> etDiagExtTPL);
						
IF etDiag <> GD.ET_Diag.Ok AND NOT xInitReactionsException THEN
	xInitReactionsException := TRUE;
	
	stInitReactionsException.sMsg := PDL.FC_MultiConcat(i_sString1 := 'InitReactionTranslationJobs - ', 
														i_sString2 := GD.FC_EtDiagToString(i_etDiag := etDiag), 
														i_sString3 := ' - ', 
														i_sString4 := TPL.FC_EtDiagExtToString(i_etDiagExt := etDiagExtTPL));
END_IF		

(*****************************************************************************************************************************************************)
(* Set exception if any exception occurred *)

fbExceptionHandler.SetException(i_xExceptionActive	:= xInitReactionsException, 
								iq_stException		:= stInitReactionsException, 
								iq_stExceptionList	:= G_stExceptionList);
					
xInitSuccessful := xInitSuccessful AND NOT xInitReactionsException;

etDiag := GD.ET_Diag.Ok;
(* End of system generated code, do not change without consulting 'Schneider Electric Automation GmbH' - otherwise you risk instability!!!*)

(* System generated code, could be modified for your application *)

(* Change of default reactions only if necessary *)
(* Examples: *)

(* A translation mode must be set for each module where the reactions should be translated *)

(* Reaction TPL.ET_Reaction.SyncStopEH in the MainMachine should act as Reaction TPL.ET_Reaction.StopEndOfCycle in BravoModule *)
// aetReactionTranslationMode[c_udiBravo] := TPL.ET_ReactionTranslationMode.Table;
// aastReactionTranslationTable[c_udiBravo,TPL.ET_Reaction.SyncStopEH].axReaction[TPL.ET_Reaction.SyncStopEH]		:= FALSE;	(* Reset old reaction *)
// aastReactionTranslationTable[c_udiBravo,TPL.ET_Reaction.SyncStopEH].axReaction[TPL.ET_Reaction.StopEndOfCycle]	:= TRUE;	(* Set new reaction *)

(* Reaction TPL.ET_Reaction.SyncStopEL in the MainMachine should act as Reaction TPL.ET_Reaction.StopEndOfCycle and TPL.ET_Reaction.MainsContactorOff in CharlyModule *)
// aetReactionTranslationMode[c_udiCharly] := TPL.ET_ReactionTranslationMode.Table;
// aastReactionTranslationTable[c_udiCharly,TPL.ET_Reaction.SyncStopEL].axReaction[TPL.ET_Reaction.SyncStopEL]			:= FALSE;	(* Reset old reaction *)
// aastReactionTranslationTable[c_udiCharly,TPL.ET_Reaction.SyncStopEL].axReaction[TPL.ET_Reaction.StopEndOfCycle]		:= TRUE;	(* Set new reaction *)
// aastReactionTranslationTable[c_udiCharly,TPL.ET_Reaction.SyncStopEL].axReaction[TPL.ET_Reaction.MainsContactorOff]	:= TRUE;	(* Set new reaction *)

(* Reaction TPL.ET_Reaction.SyncStopEL + TPL.ET_Reaction.SyncStopEH + TPL.ET_Reaction.StopEndOfCycle in the MainMachine should act as Reaction TPL.ET_Reaction.AsyncStop in AlphaModule *)
// aetReactionTranslationMode[c_udiBravo] := TPL.ET_ReactionTranslationMode.Table;
// aastReactionTranslationTable[c_udiAlpha,TPL.ET_Reaction.SyncStopEL].axReaction[TPL.ET_Reaction.SyncStopEL]			:= FALSE;	(* Reset old reaction *)
// aastReactionTranslationTable[c_udiAlpha,TPL.ET_Reaction.SyncStopEH].axReaction[TPL.ET_Reaction.SyncStopEH]			:= FALSE;	(* Reset old reaction *)
// aastReactionTranslationTable[c_udiAlpha,TPL.ET_Reaction.StopEndOfCycle].axReaction[TPL.ET_Reaction.StopEndOfCycle]	:= FALSE;	(* Reset old reaction *)
// aastReactionTranslationTable[c_udiAlpha,TPL.ET_Reaction.SyncStopEL].axReaction[TPL.ET_Reaction.AsyncStop]			:= TRUE;	(* Set new reaction *)
// aastReactionTranslationTable[c_udiAlpha,TPL.ET_Reaction.SyncStopEH].axReaction[TPL.ET_Reaction.AsyncStop]			:= TRUE;	(* Set new reaction *)
// aastReactionTranslationTable[c_udiAlpha,TPL.ET_Reaction.StopEndOfCycle].axReaction[TPL.ET_Reaction.AsyncStop]		:= TRUE;	(* Set new reaction *)

(* End of system generated code, could be modified for your application *)
END_ACTION

ACTION MainSystemFaults:
(* System generated code, do not change without consulting 'Schneider Electric Automation GmbH' - otherwise you risk instability!!! *)

IF SystemConfiguration.G_ifController <> 0 THEN
	diDiagCode := SystemConfiguration.G_ifController.DiagCode; 
	IF diDiagCode <> diDiagCode_old THEN
		diDiagCode_old	:= diDiagCode;
		stDiagSource	:= SystemConfiguration.G_ifController.DiagSource;
		IF NOT FC_ObjectTypeIsMotionAxis(i_udiObjectType := stDiagSource.udiType) THEN
			diDiagClass		:= SystemConfiguration.G_ifController.DiagClass;
			sDiagMsg		:= SystemConfiguration.G_ifController.DiagMsg;
			sInstanceName	:= 'UnknownDevice';
			SystemInterface.FC_GetObjNameByLogAddr(i_stLogAdr := stDiagSource, i_diMaxSize := SIZEOF(sInstanceName), iq_sName := sInstanceName);
			sDiagMsgExt := '';
			xSuccess := __QUERYINTERFACE(SystemConfiguration.G_ifController, ifDiagnosis);
			IF xSuccess AND (ifDiagnosis <> 0) THEN
				sDiagMsgExt := ifDiagnosis.DiagExtMsg;
			END_IF

			diDiagClass := SystemConfiguration.G_ifController.DiagClass;
			IF diDiagClass = 4 THEN
				stSystemException1.etDiag		:= GD.ET_Diag.DiagActive;
				stSystemException1.udiDiagExt	:= ET_DiagExt.SystemFatalException;								
				stSystemException1.sDiagExt		:= FC_EtDiagExtToString(stSystemException1.udiDiagExt);	
				stSystemException1.sMsg			:= PDL.FC_MultiConcat(	i_sString1 := STANDARD.CONCAT(sInstanceName, ' '),
																		i_sString2 := STANDARD.CONCAT(DINT_TO_STRING(diDiagCode), ' '), 
																		i_sString3 := STANDARD.CONCAT(sDiagMsg, ' '), 
																		i_sString4 := sDiagMsgExt);
				stSystemException1.udiExceptionNumber := TPL.FC_GenerateExceptionNumber( i_etSource := TPL.ET_ExceptionSource.System, i_udiDiagExt := DINT_TO_UDINT(diDiagCode) );
				fbExceptionHandler.SetException(i_xExceptionActive	:= TRUE,
												iq_stException		:= stSystemException1,
												iq_stExceptionList	:= G_stExceptionList);
				
			ELSIF diDiagClass = 3 THEN
				stSystemException2.etDiag		:= GD.ET_Diag.DiagActive;
				stSystemException2.udiDiagExt	:= ET_DiagExt.SystemException;				
				stSystemException2.sDiagExt		:= FC_EtDiagExtToString(stSystemException2.udiDiagExt);	
				stSystemException2.sMsg			:= PDL.FC_MultiConcat(	i_sString1 := STANDARD.CONCAT(sInstanceName, ' '),
																		i_sString2 := STANDARD.CONCAT(DINT_TO_STRING(diDiagCode), ' '), 
																		i_sString3 := STANDARD.CONCAT(sDiagMsg, ' '), 
																		i_sString4 := sDiagMsgExt);
				stSystemException2.udiExceptionNumber := TPL.FC_GenerateExceptionNumber( i_etSource := TPL.ET_ExceptionSource.System, i_udiDiagExt := DINT_TO_UDINT(diDiagCode) );
				fbExceptionHandler.SetException(i_xExceptionActive	:= TRUE,
												iq_stException		:= stSystemException2,
												iq_stExceptionList	:= G_stExceptionList);
				
			ELSIF (diDiagClass = 2 OR diDiagClass = 1) THEN
				stSystemException3.etDiag		:= GD.ET_Diag.DiagActive;
				stSystemException3.udiDiagExt	:= ET_DiagExt.SystemWarning;
				stSystemException3.sDiagExt		:= FC_EtDiagExtToString(stSystemException3.udiDiagExt);	
				stSystemException3.sMsg			:= PDL.FC_MultiConcat(	i_sString1 := STANDARD.CONCAT(sInstanceName, ' '),
																		i_sString2 := STANDARD.CONCAT(DINT_TO_STRING(diDiagCode), ' '), 
																		i_sString3 := STANDARD.CONCAT(sDiagMsg, ' '), 
																		i_sString4 := sDiagMsgExt);
				stSystemException3.udiExceptionNumber := TPL.FC_GenerateExceptionNumber( i_etSource := TPL.ET_ExceptionSource.System, i_udiDiagExt := DINT_TO_UDINT(diDiagCode) );
				fbExceptionHandler.SetException(i_xExceptionActive	:= TRUE,
												iq_stException		:= stSystemException3,
												iq_stExceptionList	:= G_stExceptionList);
			END_IF
		END_IF
	END_IF
END_IF

IF NOT xInputEmergency THEN	(* Extend logic for hardware *)

	fbExceptionHandler.SetException(i_xExceptionActive	:= TRUE,
									iq_stException		:= stEmergencyStopException,
									iq_stExceptionList	:= G_stExceptionList);
END_IF

IF etContactorControlDiag <> GD.ET_Diag.Ok THEN

	stContactorControlException.etDiag		:= etContactorControlDiag;
	stContactorControlException.udiDiagExt	:= etContactorControlDiagExt;
	stContactorControlException.sDiagExt	:= TPL.FC_EtDiagExtToString(etContactorControlDiagExt);
	stContactorControlException.sMsg		:= sContactorControlMsg;
	
	fbExceptionHandler.SetException(i_xExceptionActive	:= TRUE,
									iq_stException		:= stContactorControlException,
									iq_stExceptionList	:= G_stExceptionList);
END_IF

(* End of system generated code, do not change without consulting 'Schneider Electric Automation GmbH' - otherwise you risk instability!!! *)
END_ACTION

ACTION MainUserFaults:
(* System generated code, could be modified for your application *)
(* Test User Error *)
fbExceptionHandler.SetException(	i_xExceptionActive	:= xTestUserException2,
									iq_stException		:= stUserException2,
									iq_stExceptionList	:= G_stExceptionList,
									q_etDiag			=> etSetExceptionDiag2,
									q_etDiagExt			=> etSetExceptionDiagExt2,
									q_sMsg				=> sSetExceptionMsg2);

(* Test User Error *)
fbExceptionHandler.SetException(	i_xExceptionActive	:= xTestUserException3,
									iq_stException		:= stUserException3,
									iq_stExceptionList	:= G_stExceptionList,
									q_etDiag			=> etSetExceptionDiag3,
									q_etDiagExt			=> etSetExceptionDiagExt3,
									q_sMsg				=> sSetExceptionMsg3);
									
(* Test User Error *)
fbExceptionHandler.SetException(	i_xExceptionActive	:= xTestUserException4,
									iq_stException		:= stUserException4,
									iq_stExceptionList	:= G_stExceptionList,
									q_etDiag			=> etSetExceptionDiag4,
									q_etDiagExt			=> etSetExceptionDiagExt4,
									q_sMsg				=> sSetExceptionMsg4);
									
(* Test User Error *)
fbExceptionHandler.SetException(	i_xExceptionActive	:= xTestUserException5,
									iq_stException		:= stUserException5,
									iq_stExceptionList	:= G_stExceptionList,
									q_etDiag			=> etSetExceptionDiag5,
									q_etDiagExt			=> etSetExceptionDiagExt5,
									q_sMsg				=> sSetExceptionMsg5);
									
(* end of System generated code, could be modified for your application *)
END_ACTION

METHOD AssignCarriers
VAR_INPUT
END_VAR
//--- Assign the Segments here.
{IF defined (variable:MC_Carrier_1)}
	stMulticarrierModule.i_aifMulticarrierCarriers[1]		:= MC_Carrier_1;
{END_IF}
{IF defined (variable:MC_Carrier_2)}
	stMulticarrierModule.i_aifMulticarrierCarriers[2]		:= MC_Carrier_2;
{END_IF}
{IF defined (variable:MC_Carrier_3)}
	stMulticarrierModule.i_aifMulticarrierCarriers[3]		:= MC_Carrier_3;
{END_IF}
{IF defined (variable:MC_Carrier_4)}
	stMulticarrierModule.i_aifMulticarrierCarriers[4]		:= MC_Carrier_4;
{END_IF}
{IF defined (variable:MC_Carrier_5)}
	stMulticarrierModule.i_aifMulticarrierCarriers[5]		:= MC_Carrier_5;
{END_IF}
{IF defined (variable:MC_Carrier_6)}
	stMulticarrierModule.i_aifMulticarrierCarriers[6]		:= MC_Carrier_6;
{END_IF}
{IF defined (variable:MC_Carrier_7)}
	stMulticarrierModule.i_aifMulticarrierCarriers[7]		:= MC_Carrier_7;
{END_IF}
{IF defined (variable:MC_Carrier_8)}
	stMulticarrierModule.i_aifMulticarrierCarriers[8]		:= MC_Carrier_8;
{END_IF}
{IF defined (variable:MC_Carrier_9)}
	stMulticarrierModule.i_aifMulticarrierCarriers[9]		:= MC_Carrier_9;
{END_IF}
{IF defined (variable:MC_Carrier_10)}
	stMulticarrierModule.i_aifMulticarrierCarriers[10]		:= MC_Carrier_10;
{END_IF}
{IF defined (variable:MC_Carrier_11)}
	stMulticarrierModule.i_aifMulticarrierCarriers[11]		:= MC_Carrier_11;
{END_IF}
{IF defined (variable:MC_Carrier_12)}
	stMulticarrierModule.i_aifMulticarrierCarriers[12]		:= MC_Carrier_12;
{END_IF}
{IF defined (variable:MC_Carrier_13)}
	stMulticarrierModule.i_aifMulticarrierCarriers[13]		:= MC_Carrier_13;
{END_IF}
{IF defined (variable:MC_Carrier_14)}
	stMulticarrierModule.i_aifMulticarrierCarriers[14]		:= MC_Carrier_14;
{END_IF}
{IF defined (variable:MC_Carrier_15)}
	stMulticarrierModule.i_aifMulticarrierCarriers[15]		:= MC_Carrier_15;
{END_IF}
{IF defined (variable:MC_Carrier_16)}
	stMulticarrierModule.i_aifMulticarrierCarriers[16]		:= MC_Carrier_16;
{END_IF}
{IF defined (variable:MC_Carrier_17)}
 	stMulticarrierModule.i_aifMulticarrierCarriers[17]		:= MC_Carrier_17;
 {END_IF}
 {IF defined (variable:MC_Carrier_18)}
 	stMulticarrierModule.i_aifMulticarrierCarriers[18]		:= MC_Carrier_18;
 {END_IF}
 {IF defined (variable:MC_Carrier_19)}
 	stMulticarrierModule.i_aifMulticarrierCarriers[19]		:= MC_Carrier_19;
 {END_IF}
 {IF defined (variable:MC_Carrier_20)}
 	stMulticarrierModule.i_aifMulticarrierCarriers[20]		:= MC_Carrier_20;
 {END_IF}
 {IF defined (variable:MC_Carrier_21)}
	stMulticarrierModule.i_aifMulticarrierCarriers[21]		:= MC_Carrier_21;
{END_IF}
{IF defined (variable:MC_Carrier_22)}
	stMulticarrierModule.i_aifMulticarrierCarriers[22]		:= MC_Carrier_22;
{END_IF}
{IF defined (variable:MC_Carrier_23)}
	stMulticarrierModule.i_aifMulticarrierCarriers[23]		:= MC_Carrier_23;
{END_IF}
{IF defined (variable:MC_Carrier_24)}
	stMulticarrierModule.i_aifMulticarrierCarriers[24]		:= MC_Carrier_24;
{END_IF}
{IF defined (variable:MC_Carrier_25)}
	stMulticarrierModule.i_aifMulticarrierCarriers[25]		:= MC_Carrier_25;
{END_IF}
{IF defined (variable:MC_Carrier_26)}
	stMulticarrierModule.i_aifMulticarrierCarriers[26]		:= MC_Carrier_26;
{END_IF}
{IF defined (variable:MC_Carrier_27)}
 	stMulticarrierModule.i_aifMulticarrierCarriers[27]		:= MC_Carrier_27;
 {END_IF}
 {IF defined (variable:MC_Carrier_28)}
 	stMulticarrierModule.i_aifMulticarrierCarriers[28]		:= MC_Carrier_28;
 {END_IF}
 {IF defined (variable:MC_Carrier_29)}
 	stMulticarrierModule.i_aifMulticarrierCarriers[29]		:= MC_Carrier_29;
 {END_IF}
 {IF defined (variable:MC_Carrier_30)}
 	stMulticarrierModule.i_aifMulticarrierCarriers[30]		:= MC_Carrier_30;
 {END_IF}
 {IF defined (variable:MC_Carrier_31)}
	stMulticarrierModule.i_aifMulticarrierCarriers[31]		:= MC_Carrier_31;
{END_IF}
{IF defined (variable:MC_Carrier_32)}
	stMulticarrierModule.i_aifMulticarrierCarriers[32]		:= MC_Carrier_32;
{END_IF}
{IF defined (variable:MC_Carrier_33)}
	stMulticarrierModule.i_aifMulticarrierCarriers[33]		:= MC_Carrier_33;
{END_IF}
{IF defined (variable:MC_Carrier_34)}
	stMulticarrierModule.i_aifMulticarrierCarriers[34]		:= MC_Carrier_34;
{END_IF}
{IF defined (variable:MC_Carrier_35)}
	stMulticarrierModule.i_aifMulticarrierCarriers[35]		:= MC_Carrier_35;
{END_IF}
{IF defined (variable:MC_Carrier_36)}
	stMulticarrierModule.i_aifMulticarrierCarriers[36]		:= MC_Carrier_36;
{END_IF}
{IF defined (variable:MC_Carrier_37)}
 	stMulticarrierModule.i_aifMulticarrierCarriers[37]		:= MC_Carrier_37;
 {END_IF}
 {IF defined (variable:MC_Carrier_38)}
 	stMulticarrierModule.i_aifMulticarrierCarriers[38]		:= MC_Carrier_38;
 {END_IF}
 {IF defined (variable:MC_Carrier_39)}
 	stMulticarrierModule.i_aifMulticarrierCarriers[39]		:= MC_Carrier_39;
 {END_IF} 
 {IF defined (variable:MC_Carrier_40)}
 	stMulticarrierModule.i_aifMulticarrierCarriers[40]		:= MC_Carrier_40;
 {END_IF}
 {IF defined (variable:MC_Carrier_41)}
	stMulticarrierModule.i_aifMulticarrierCarriers[41]		:= MC_Carrier_41;
{END_IF}
{IF defined (variable:MC_Carrier_42)}
	stMulticarrierModule.i_aifMulticarrierCarriers[42]		:= MC_Carrier_42;
{END_IF}
{IF defined (variable:MC_Carrier_43)}
	stMulticarrierModule.i_aifMulticarrierCarriers[43]		:= MC_Carrier_43;
{END_IF}
{IF defined (variable:MC_Carrier_44)}
	stMulticarrierModule.i_aifMulticarrierCarriers[44]		:= MC_Carrier_44;
{END_IF}
{IF defined (variable:MC_Carrier_45)}
	stMulticarrierModule.i_aifMulticarrierCarriers[45]		:= MC_Carrier_45;
{END_IF}
{IF defined (variable:MC_Carrier_46)}
	stMulticarrierModule.i_aifMulticarrierCarriers[46]		:= MC_Carrier_46;
{END_IF}
{IF defined (variable:MC_Carrier_47)}
 	stMulticarrierModule.i_aifMulticarrierCarriers[47]		:= MC_Carrier_47;
 {END_IF}
 {IF defined (variable:MC_Carrier_48)}
 	stMulticarrierModule.i_aifMulticarrierCarriers[48]		:= MC_Carrier_48;
 {END_IF}
 {IF defined (variable:MC_Carrier_49)}
 	stMulticarrierModule.i_aifMulticarrierCarriers[49]		:= MC_Carrier_49;
 {END_IF}
  {IF defined (variable:MC_Carrier_50)}
 	stMulticarrierModule.i_aifMulticarrierCarriers[50]		:= MC_Carrier_50;
 {END_IF}
 {IF defined (variable:MC_Carrier_51)}
	stMulticarrierModule.i_aifMulticarrierCarriers[51]		:= MC_Carrier_51;
{END_IF}
{IF defined (variable:MC_Carrier_52)}
	stMulticarrierModule.i_aifMulticarrierCarriers[52]		:= MC_Carrier_52;
{END_IF}
{IF defined (variable:MC_Carrier_53)}
	stMulticarrierModule.i_aifMulticarrierCarriers[53]		:= MC_Carrier_53;
{END_IF}
{IF defined (variable:MC_Carrier_54)}
	stMulticarrierModule.i_aifMulticarrierCarriers[54]		:= MC_Carrier_54;
{END_IF}
{IF defined (variable:MC_Carrier_55)}
	stMulticarrierModule.i_aifMulticarrierCarriers[55]		:= MC_Carrier_55;
{END_IF}
{IF defined (variable:MC_Carrier_56)}
	stMulticarrierModule.i_aifMulticarrierCarriers[56]		:= MC_Carrier_56;
{END_IF}
{IF defined (variable:MC_Carrier_57)}
 	stMulticarrierModule.i_aifMulticarrierCarriers[57]		:= MC_Carrier_57;
 {END_IF}
 {IF defined (variable:MC_Carrier_58)}
 	stMulticarrierModule.i_aifMulticarrierCarriers[58]		:= MC_Carrier_58;
 {END_IF}
 {IF defined (variable:MC_Carrier_59)}
 	stMulticarrierModule.i_aifMulticarrierCarriers[59]		:= MC_Carrier_59;
 {END_IF}
  {IF defined (variable:MC_Carrier_60)}
 	stMulticarrierModule.i_aifMulticarrierCarriers[60]		:= MC_Carrier_60;
 {END_IF}
 {IF defined (variable:MC_Carrier_61)}
	stMulticarrierModule.i_aifMulticarrierCarriers[61]		:= MC_Carrier_61;
{END_IF}
{IF defined (variable:MC_Carrier_62)}
	stMulticarrierModule.i_aifMulticarrierCarriers[62]		:= MC_Carrier_62;
{END_IF}
{IF defined (variable:MC_Carrier_63)}
	stMulticarrierModule.i_aifMulticarrierCarriers[63]		:= MC_Carrier_63;
{END_IF}
{IF defined (variable:MC_Carrier_64)}
	stMulticarrierModule.i_aifMulticarrierCarriers[64]		:= MC_Carrier_64;
{END_IF}
{IF defined (variable:MC_Carrier_65)}
	stMulticarrierModule.i_aifMulticarrierCarriers[65]		:= MC_Carrier_65;
{END_IF}
{IF defined (variable:MC_Carrier_66)}
	stMulticarrierModule.i_aifMulticarrierCarriers[66]		:= MC_Carrier_66;
{END_IF}
{IF defined (variable:MC_Carrier_67)}
 	stMulticarrierModule.i_aifMulticarrierCarriers[67]		:= MC_Carrier_67;
 {END_IF}
 {IF defined (variable:MC_Carrier_68)}
 	stMulticarrierModule.i_aifMulticarrierCarriers[68]		:= MC_Carrier_68;
 {END_IF}
 {IF defined (variable:MC_Carrier_69)}
 	stMulticarrierModule.i_aifMulticarrierCarriers[69]		:= MC_Carrier_69;
 {END_IF}
  {IF defined (variable:MC_Carrier_70)}
 	stMulticarrierModule.i_aifMulticarrierCarriers[70]		:= MC_Carrier_70;
 {END_IF}
 {IF defined (variable:MC_Carrier_71)}
	stMulticarrierModule.i_aifMulticarrierCarriers[71]		:= MC_Carrier_71;
{END_IF}
{IF defined (variable:MC_Carrier_72)}
	stMulticarrierModule.i_aifMulticarrierCarriers[72]		:= MC_Carrier_72;
{END_IF}
{IF defined (variable:MC_Carrier_73)}
	stMulticarrierModule.i_aifMulticarrierCarriers[73]		:= MC_Carrier_73;
{END_IF}
{IF defined (variable:MC_Carrier_74)}
	stMulticarrierModule.i_aifMulticarrierCarriers[74]		:= MC_Carrier_74;
{END_IF}
{IF defined (variable:MC_Carrier_75)}
	stMulticarrierModule.i_aifMulticarrierCarriers[75]		:= MC_Carrier_75;
{END_IF}
{IF defined (variable:MC_Carrier_76)}
	stMulticarrierModule.i_aifMulticarrierCarriers[76]		:= MC_Carrier_76;
{END_IF}
{IF defined (variable:MC_Carrier_77)}
 	stMulticarrierModule.i_aifMulticarrierCarriers[77]		:= MC_Carrier_77;
 {END_IF}
 {IF defined (variable:MC_Carrier_78)}
 	stMulticarrierModule.i_aifMulticarrierCarriers[78]		:= MC_Carrier_78;
 {END_IF}
 {IF defined (variable:MC_Carrier_79)}
 	stMulticarrierModule.i_aifMulticarrierCarriers[79]		:= MC_Carrier_79;
 {END_IF}
  {IF defined (variable:MC_Carrier_80)}
 	stMulticarrierModule.i_aifMulticarrierCarriers[80]		:= MC_Carrier_80;
 {END_IF}
 {IF defined (variable:MC_Carrier_81)}
	stMulticarrierModule.i_aifMulticarrierCarriers[81]		:= MC_Carrier_81;
{END_IF}
{IF defined (variable:MC_Carrier_82)}
	stMulticarrierModule.i_aifMulticarrierCarriers[82]		:= MC_Carrier_82;
{END_IF}
{IF defined (variable:MC_Carrier_83)}
	stMulticarrierModule.i_aifMulticarrierCarriers[83]		:= MC_Carrier_83;
{END_IF}
{IF defined (variable:MC_Carrier_84)}
	stMulticarrierModule.i_aifMulticarrierCarriers[84]		:= MC_Carrier_84;
{END_IF}
{IF defined (variable:MC_Carrier_85)}
	stMulticarrierModule.i_aifMulticarrierCarriers[85]		:= MC_Carrier_85;
{END_IF}
{IF defined (variable:MC_Carrier_86)}
	stMulticarrierModule.i_aifMulticarrierCarriers[86]		:= MC_Carrier_86;
{END_IF}
{IF defined (variable:MC_Carrier_87)}
 	stMulticarrierModule.i_aifMulticarrierCarriers[87]		:= MC_Carrier_87;
 {END_IF}
 {IF defined (variable:MC_Carrier_88)}
 	stMulticarrierModule.i_aifMulticarrierCarriers[88]		:= MC_Carrier_88;
 {END_IF}
 {IF defined (variable:MC_Carrier_89)}
 	stMulticarrierModule.i_aifMulticarrierCarriers[89]		:= MC_Carrier_89;
 {END_IF}
  {IF defined (variable:MC_Carrier_90)}
 	stMulticarrierModule.i_aifMulticarrierCarriers[90]		:= MC_Carrier_90;
 {END_IF}
 {IF defined (variable:MC_Carrier_91)}
	stMulticarrierModule.i_aifMulticarrierCarriers[91]		:= MC_Carrier_91;
{END_IF}
{IF defined (variable:MC_Carrier_92)}
	stMulticarrierModule.i_aifMulticarrierCarriers[92]		:= MC_Carrier_92;
{END_IF}
{IF defined (variable:MC_Carrier_93)}
	stMulticarrierModule.i_aifMulticarrierCarriers[93]		:= MC_Carrier_93;
{END_IF}
{IF defined (variable:MC_Carrier_94)}
	stMulticarrierModule.i_aifMulticarrierCarriers[94]		:= MC_Carrier_94;
{END_IF}
{IF defined (variable:MC_Carrier_95)}
	stMulticarrierModule.i_aifMulticarrierCarriers[95]		:= MC_Carrier_95;
{END_IF}
{IF defined (variable:MC_Carrier_96)}
	stMulticarrierModule.i_aifMulticarrierCarriers[96]		:= MC_Carrier_96;
{END_IF}
{IF defined (variable:MC_Carrier_97)}
 	stMulticarrierModule.i_aifMulticarrierCarriers[97]		:= MC_Carrier_97;
 {END_IF}
 {IF defined (variable:MC_Carrier_98)}
 	stMulticarrierModule.i_aifMulticarrierCarriers[98]		:= MC_Carrier_98;
 {END_IF}
 {IF defined (variable:MC_Carrier_99)}
 	stMulticarrierModule.i_aifMulticarrierCarriers[99]		:= MC_Carrier_99;
 {END_IF}
  {IF defined (variable:MC_Carrier_100)}
 	stMulticarrierModule.i_aifMulticarrierCarriers[100]		:= MC_Carrier_100;
 {END_IF}
 {IF defined (variable:MC_Carrier_101)}
	stMulticarrierModule.i_aifMulticarrierCarriers[101]		:= MC_Carrier_101;
{END_IF}
{IF defined (variable:MC_Carrier_102)}
	stMulticarrierModule.i_aifMulticarrierCarriers[102]		:= MC_Carrier_102;
{END_IF}
{IF defined (variable:MC_Carrier_103)}
	stMulticarrierModule.i_aifMulticarrierCarriers[103]		:= MC_Carrier_103;
{END_IF}
{IF defined (variable:MC_Carrier_104)}
	stMulticarrierModule.i_aifMulticarrierCarriers[104]		:= MC_Carrier_104;
{END_IF}
{IF defined (variable:MC_Carrier_105)}
	stMulticarrierModule.i_aifMulticarrierCarriers[105]		:= MC_Carrier_105;
{END_IF}
{IF defined (variable:MC_Carrier_106)}
	stMulticarrierModule.i_aifMulticarrierCarriers[106]		:= MC_Carrier_106;
{END_IF}
{IF defined (variable:MC_Carrier_107)}
	stMulticarrierModule.i_aifMulticarrierCarriers[107]		:= MC_Carrier_107;
{END_IF}
{IF defined (variable:MC_Carrier_108)}
	stMulticarrierModule.i_aifMulticarrierCarriers[108]		:= MC_Carrier_108;
{END_IF}
{IF defined (variable:MC_Carrier_109)}
	stMulticarrierModule.i_aifMulticarrierCarriers[109]		:= MC_Carrier_109;
{END_IF} 
{IF defined (variable:MC_Carrier_110)}
 	stMulticarrierModule.i_aifMulticarrierCarriers[110]		:= MC_Carrier_110;
{END_IF}
 {IF defined (variable:MC_Carrier_111)}
	stMulticarrierModule.i_aifMulticarrierCarriers[111]		:= MC_Carrier_111;
{END_IF}
{IF defined (variable:MC_Carrier_112)}
	stMulticarrierModule.i_aifMulticarrierCarriers[112]		:= MC_Carrier_112;
{END_IF}
{IF defined (variable:MC_Carrier_113)}
	stMulticarrierModule.i_aifMulticarrierCarriers[113]		:= MC_Carrier_113;
{END_IF}
{IF defined (variable:MC_Carrier_114)}
	stMulticarrierModule.i_aifMulticarrierCarriers[114]		:= MC_Carrier_114;
{END_IF}
{IF defined (variable:MC_Carrier_115)}
	stMulticarrierModule.i_aifMulticarrierCarriers[115]		:= MC_Carrier_115;
{END_IF}
{IF defined (variable:MC_Carrier_116)}
	stMulticarrierModule.i_aifMulticarrierCarriers[116]		:= MC_Carrier_116;
{END_IF}
{IF defined (variable:MC_Carrier_117)}
	stMulticarrierModule.i_aifMulticarrierCarriers[117]		:= MC_Carrier_117;
{END_IF}
{IF defined (variable:MC_Carrier_118)}
	stMulticarrierModule.i_aifMulticarrierCarriers[118]		:= MC_Carrier_118;
{END_IF}
{IF defined (variable:MC_Carrier_119)}
	stMulticarrierModule.i_aifMulticarrierCarriers[119]		:= MC_Carrier_119;
{END_IF}  
{IF defined (variable:MC_Carrier_120)}
 	stMulticarrierModule.i_aifMulticarrierCarriers[120]		:= MC_Carrier_120;
{END_IF}
 {IF defined (variable:MC_Carrier_121)}
	stMulticarrierModule.i_aifMulticarrierCarriers[121]		:= MC_Carrier_121;
{END_IF}
{IF defined (variable:MC_Carrier_122)}
	stMulticarrierModule.i_aifMulticarrierCarriers[122]		:= MC_Carrier_122;
{END_IF}
{IF defined (variable:MC_Carrier_123)}
	stMulticarrierModule.i_aifMulticarrierCarriers[123]		:= MC_Carrier_123;
{END_IF}
{IF defined (variable:MC_Carrier_124)}
	stMulticarrierModule.i_aifMulticarrierCarriers[124]		:= MC_Carrier_124;
{END_IF}
{IF defined (variable:MC_Carrier_125)}
	stMulticarrierModule.i_aifMulticarrierCarriers[125]		:= MC_Carrier_125;
{END_IF}
{IF defined (variable:MC_Carrier_126)}
	stMulticarrierModule.i_aifMulticarrierCarriers[126]		:= MC_Carrier_126;
{END_IF}
{IF defined (variable:MC_Carrier_127)}
	stMulticarrierModule.i_aifMulticarrierCarriers[127]		:= MC_Carrier_127;
{END_IF}
{IF defined (variable:MC_Carrier_128)}
	stMulticarrierModule.i_aifMulticarrierCarriers[128]		:= MC_Carrier_128;
{END_IF}
{IF defined (variable:MC_Carrier_129)}
	stMulticarrierModule.i_aifMulticarrierCarriers[129]		:= MC_Carrier_129;
{END_IF}   
{IF defined (variable:MC_Carrier_130)}
 	stMulticarrierModule.i_aifMulticarrierCarriers[130]		:= MC_Carrier_130;
{END_IF}
 {IF defined (variable:MC_Carrier_131)}
	stMulticarrierModule.i_aifMulticarrierCarriers[131]		:= MC_Carrier_131;
{END_IF}
{IF defined (variable:MC_Carrier_132)}
	stMulticarrierModule.i_aifMulticarrierCarriers[132]		:= MC_Carrier_132;
{END_IF}
{IF defined (variable:MC_Carrier_133)}
	stMulticarrierModule.i_aifMulticarrierCarriers[133]		:= MC_Carrier_133;
{END_IF}
{IF defined (variable:MC_Carrier_134)}
	stMulticarrierModule.i_aifMulticarrierCarriers[134]		:= MC_Carrier_134;
{END_IF}
{IF defined (variable:MC_Carrier_135)}
	stMulticarrierModule.i_aifMulticarrierCarriers[135]		:= MC_Carrier_135;
{END_IF}
{IF defined (variable:MC_Carrier_136)}
	stMulticarrierModule.i_aifMulticarrierCarriers[136]		:= MC_Carrier_136;
{END_IF}
{IF defined (variable:MC_Carrier_137)}
	stMulticarrierModule.i_aifMulticarrierCarriers[137]		:= MC_Carrier_137;
{END_IF}
{IF defined (variable:MC_Carrier_138)}
	stMulticarrierModule.i_aifMulticarrierCarriers[138]		:= MC_Carrier_138;
{END_IF}
{IF defined (variable:MC_Carrier_139)}
	stMulticarrierModule.i_aifMulticarrierCarriers[139]		:= MC_Carrier_139;
{END_IF}   
{IF defined (variable:MC_Carrier_140)}
 	stMulticarrierModule.i_aifMulticarrierCarriers[140]		:= MC_Carrier_140;
{END_IF}
 {IF defined (variable:MC_Carrier_141)}
	stMulticarrierModule.i_aifMulticarrierCarriers[141]		:= MC_Carrier_141;
{END_IF}
{IF defined (variable:MC_Carrier_142)}
	stMulticarrierModule.i_aifMulticarrierCarriers[142]		:= MC_Carrier_142;
{END_IF}
{IF defined (variable:MC_Carrier_143)}
	stMulticarrierModule.i_aifMulticarrierCarriers[143]		:= MC_Carrier_143;
{END_IF}
{IF defined (variable:MC_Carrier_144)}
	stMulticarrierModule.i_aifMulticarrierCarriers[144]		:= MC_Carrier_144;
{END_IF}
{IF defined (variable:MC_Carrier_145)}
	stMulticarrierModule.i_aifMulticarrierCarriers[145]		:= MC_Carrier_145;
{END_IF}
{IF defined (variable:MC_Carrier_146)}
	stMulticarrierModule.i_aifMulticarrierCarriers[146]		:= MC_Carrier_146;
{END_IF}
{IF defined (variable:MC_Carrier_147)}
	stMulticarrierModule.i_aifMulticarrierCarriers[147]		:= MC_Carrier_147;
{END_IF}
{IF defined (variable:MC_Carrier_148)}
	stMulticarrierModule.i_aifMulticarrierCarriers[148]		:= MC_Carrier_148;
{END_IF}
{IF defined (variable:MC_Carrier_149)}
	stMulticarrierModule.i_aifMulticarrierCarriers[149]		:= MC_Carrier_149;
{END_IF}   
{IF defined (variable:MC_Carrier_150)}
 	stMulticarrierModule.i_aifMulticarrierCarriers[150]		:= MC_Carrier_150;
{END_IF}
END_METHOD

METHOD AssignSegments
VAR_INPUT
END_VAR
//--- Assign the Segments here.
{IF defined (variable:MC_Segment_1)}
	stMulticarrierModule.i_aifMulticarrierSegments[1]		:= MC_Segment_1;
{END_IF}
{IF defined (variable:MC_Segment_2)}
	stMulticarrierModule.i_aifMulticarrierSegments[2]		:= MC_Segment_2;
{END_IF}
{IF defined (variable:MC_Segment_3)}
	stMulticarrierModule.i_aifMulticarrierSegments[3]		:= MC_Segment_3;
{END_IF}
{IF defined (variable:MC_Segment_4)}
	stMulticarrierModule.i_aifMulticarrierSegments[4]		:= MC_Segment_4;
{END_IF}
{IF defined (variable:MC_Segment_5)}
	stMulticarrierModule.i_aifMulticarrierSegments[5]		:= MC_Segment_5;
{END_IF}
{IF defined (variable:MC_Segment_6)}
	stMulticarrierModule.i_aifMulticarrierSegments[6]		:= MC_Segment_6;
{END_IF}
{IF defined (variable:MC_Segment_7)}
	stMulticarrierModule.i_aifMulticarrierSegments[7]		:= MC_Segment_7;
{END_IF}
{IF defined (variable:MC_Segment_8)}
	stMulticarrierModule.i_aifMulticarrierSegments[8]		:= MC_Segment_8;
{END_IF}
{IF defined (variable:MC_Segment_9)}
	stMulticarrierModule.i_aifMulticarrierSegments[9]		:= MC_Segment_9;
{END_IF}
{IF defined (variable:MC_Segment_10)}
	stMulticarrierModule.i_aifMulticarrierSegments[10]		:= MC_Segment_10;
{END_IF}
{IF defined (variable:MC_Segment_11)}
	stMulticarrierModule.i_aifMulticarrierSegments[11]		:= MC_Segment_11;
{END_IF}
{IF defined (variable:MC_Segment_12)}
	stMulticarrierModule.i_aifMulticarrierSegments[12]		:= MC_Segment_12;
{END_IF}
{IF defined (variable:MC_Segment_13)}
	stMulticarrierModule.i_aifMulticarrierSegments[13]		:= MC_Segment_13;
{END_IF}
{IF defined (variable:MC_Segment_14)}
	stMulticarrierModule.i_aifMulticarrierSegments[14]		:= MC_Segment_14;
{END_IF}
{IF defined (variable:MC_Segment_15)}
	stMulticarrierModule.i_aifMulticarrierSegments[15]		:= MC_Segment_15;
{END_IF}
{IF defined (variable:MC_Segment_16)}
	stMulticarrierModule.i_aifMulticarrierSegments[16]		:= MC_Segment_16;
{END_IF}
{IF defined (variable:MC_Segment_17)}
 	stMulticarrierModule.i_aifMulticarrierSegments[17]		:= MC_Segment_17;
 {END_IF}
 {IF defined (variable:MC_Segment_18)}
 	stMulticarrierModule.i_aifMulticarrierSegments[18]		:= MC_Segment_18;
 {END_IF}
 {IF defined (variable:MC_Segment_19)}
 	stMulticarrierModule.i_aifMulticarrierSegments[19]		:= MC_Segment_19;
 {END_IF}
 {IF defined (variable:MC_Segment_20)}
 	stMulticarrierModule.i_aifMulticarrierSegments[20]		:= MC_Segment_20;
 {END_IF}
 {IF defined (variable:MC_Segment_21)}
	stMulticarrierModule.i_aifMulticarrierSegments[21]		:= MC_Segment_21;
{END_IF}
{IF defined (variable:MC_Segment_22)}
	stMulticarrierModule.i_aifMulticarrierSegments[22]		:= MC_Segment_22;
{END_IF}
{IF defined (variable:MC_Segment_23)}
	stMulticarrierModule.i_aifMulticarrierSegments[23]		:= MC_Segment_23;
{END_IF}
{IF defined (variable:MC_Segment_24)}
	stMulticarrierModule.i_aifMulticarrierSegments[24]		:= MC_Segment_24;
{END_IF}
{IF defined (variable:MC_Segment_25)}
	stMulticarrierModule.i_aifMulticarrierSegments[25]		:= MC_Segment_25;
{END_IF}
{IF defined (variable:MC_Segment_26)}
	stMulticarrierModule.i_aifMulticarrierSegments[26]		:= MC_Segment_26;
{END_IF}
{IF defined (variable:MC_Segment_27)}
 	stMulticarrierModule.i_aifMulticarrierSegments[27]		:= MC_Segment_27;
 {END_IF}
 {IF defined (variable:MC_Segment_28)}
 	stMulticarrierModule.i_aifMulticarrierSegments[28]		:= MC_Segment_28;
 {END_IF}
 {IF defined (variable:MC_Segment_29)}
 	stMulticarrierModule.i_aifMulticarrierSegments[29]		:= MC_Segment_29;
 {END_IF}
 {IF defined (variable:MC_Segment_30)}
 	stMulticarrierModule.i_aifMulticarrierSegments[30]		:= MC_Segment_30;
 {END_IF}
 {IF defined (variable:MC_Segment_31)}
	stMulticarrierModule.i_aifMulticarrierSegments[31]		:= MC_Segment_31;
{END_IF}
{IF defined (variable:MC_Segment_32)}
	stMulticarrierModule.i_aifMulticarrierSegments[32]		:= MC_Segment_32;
{END_IF}
{IF defined (variable:MC_Segment_33)}
	stMulticarrierModule.i_aifMulticarrierSegments[33]		:= MC_Segment_33;
{END_IF}
{IF defined (variable:MC_Segment_34)}
	stMulticarrierModule.i_aifMulticarrierSegments[34]		:= MC_Segment_34;
{END_IF}
{IF defined (variable:MC_Segment_35)}
	stMulticarrierModule.i_aifMulticarrierSegments[35]		:= MC_Segment_35;
{END_IF}
{IF defined (variable:MC_Segment_36)}
	stMulticarrierModule.i_aifMulticarrierSegments[36]		:= MC_Segment_36;
{END_IF}
{IF defined (variable:MC_Segment_37)}
 	stMulticarrierModule.i_aifMulticarrierSegments[37]		:= MC_Segment_37;
 {END_IF}
 {IF defined (variable:MC_Segment_38)}
 	stMulticarrierModule.i_aifMulticarrierSegments[38]		:= MC_Segment_38;
 {END_IF}
 {IF defined (variable:MC_Segment_39)}
 	stMulticarrierModule.i_aifMulticarrierSegments[39]		:= MC_Segment_39;
 {END_IF} 
 {IF defined (variable:MC_Segment_40)}
 	stMulticarrierModule.i_aifMulticarrierSegments[40]		:= MC_Segment_40;
 {END_IF}
 {IF defined (variable:MC_Segment_41)}
	stMulticarrierModule.i_aifMulticarrierSegments[41]		:= MC_Segment_41;
{END_IF}
{IF defined (variable:MC_Segment_42)}
	stMulticarrierModule.i_aifMulticarrierSegments[42]		:= MC_Segment_42;
{END_IF}
{IF defined (variable:MC_Segment_43)}
	stMulticarrierModule.i_aifMulticarrierSegments[43]		:= MC_Segment_43;
{END_IF}
{IF defined (variable:MC_Segment_44)}
	stMulticarrierModule.i_aifMulticarrierSegments[44]		:= MC_Segment_44;
{END_IF}
{IF defined (variable:MC_Segment_45)}
	stMulticarrierModule.i_aifMulticarrierSegments[45]		:= MC_Segment_45;
{END_IF}
{IF defined (variable:MC_Segment_46)}
	stMulticarrierModule.i_aifMulticarrierSegments[46]		:= MC_Segment_46;
{END_IF}
{IF defined (variable:MC_Segment_47)}
 	stMulticarrierModule.i_aifMulticarrierSegments[47]		:= MC_Segment_47;
 {END_IF}
 {IF defined (variable:MC_Segment_48)}
 	stMulticarrierModule.i_aifMulticarrierSegments[48]		:= MC_Segment_48;
 {END_IF}
 {IF defined (variable:MC_Segment_49)}
 	stMulticarrierModule.i_aifMulticarrierSegments[49]		:= MC_Segment_49;
 {END_IF}
  {IF defined (variable:MC_Segment_50)}
 	stMulticarrierModule.i_aifMulticarrierSegments[50]		:= MC_Segment_50;
 {END_IF}
 {IF defined (variable:MC_Segment_51)}
	stMulticarrierModule.i_aifMulticarrierSegments[51]		:= MC_Segment_51;
{END_IF}
{IF defined (variable:MC_Segment_52)}
	stMulticarrierModule.i_aifMulticarrierSegments[52]		:= MC_Segment_52;
{END_IF}
{IF defined (variable:MC_Segment_53)}
	stMulticarrierModule.i_aifMulticarrierSegments[53]		:= MC_Segment_53;
{END_IF}
{IF defined (variable:MC_Segment_54)}
	stMulticarrierModule.i_aifMulticarrierSegments[54]		:= MC_Segment_54;
{END_IF}
{IF defined (variable:MC_Segment_55)}
	stMulticarrierModule.i_aifMulticarrierSegments[55]		:= MC_Segment_55;
{END_IF}
{IF defined (variable:MC_Segment_56)}
	stMulticarrierModule.i_aifMulticarrierSegments[56]		:= MC_Segment_56;
{END_IF}
{IF defined (variable:MC_Segment_57)}
 	stMulticarrierModule.i_aifMulticarrierSegments[57]		:= MC_Segment_57;
 {END_IF}
 {IF defined (variable:MC_Segment_58)}
 	stMulticarrierModule.i_aifMulticarrierSegments[58]		:= MC_Segment_58;
 {END_IF}
 {IF defined (variable:MC_Segment_59)}
 	stMulticarrierModule.i_aifMulticarrierSegments[59]		:= MC_Segment_59;
 {END_IF}
  {IF defined (variable:MC_Segment_60)}
 	stMulticarrierModule.i_aifMulticarrierSegments[60]		:= MC_Segment_60;
 {END_IF}
 {IF defined (variable:MC_Segment_61)}
	stMulticarrierModule.i_aifMulticarrierSegments[61]		:= MC_Segment_61;
{END_IF}
{IF defined (variable:MC_Segment_62)}
	stMulticarrierModule.i_aifMulticarrierSegments[62]		:= MC_Segment_62;
{END_IF}
{IF defined (variable:MC_Segment_63)}
	stMulticarrierModule.i_aifMulticarrierSegments[63]		:= MC_Segment_63;
{END_IF}
{IF defined (variable:MC_Segment_64)}
	stMulticarrierModule.i_aifMulticarrierSegments[64]		:= MC_Segment_64;
{END_IF}
{IF defined (variable:MC_Segment_65)}
	stMulticarrierModule.i_aifMulticarrierSegments[65]		:= MC_Segment_65;
{END_IF}
{IF defined (variable:MC_Segment_66)}
	stMulticarrierModule.i_aifMulticarrierSegments[66]		:= MC_Segment_66;
{END_IF}
{IF defined (variable:MC_Segment_67)}
 	stMulticarrierModule.i_aifMulticarrierSegments[67]		:= MC_Segment_67;
 {END_IF}
 {IF defined (variable:MC_Segment_68)}
 	stMulticarrierModule.i_aifMulticarrierSegments[68]		:= MC_Segment_68;
 {END_IF}
 {IF defined (variable:MC_Segment_69)}
 	stMulticarrierModule.i_aifMulticarrierSegments[69]		:= MC_Segment_69;
 {END_IF}
  {IF defined (variable:MC_Segment_70)}
 	stMulticarrierModule.i_aifMulticarrierSegments[70]		:= MC_Segment_70;
 {END_IF}
 {IF defined (variable:MC_Segment_71)}
	stMulticarrierModule.i_aifMulticarrierSegments[71]		:= MC_Segment_71;
{END_IF}
{IF defined (variable:MC_Segment_72)}
	stMulticarrierModule.i_aifMulticarrierSegments[72]		:= MC_Segment_72;
{END_IF}
{IF defined (variable:MC_Segment_73)}
	stMulticarrierModule.i_aifMulticarrierSegments[73]		:= MC_Segment_73;
{END_IF}
{IF defined (variable:MC_Segment_74)}
	stMulticarrierModule.i_aifMulticarrierSegments[74]		:= MC_Segment_74;
{END_IF}
{IF defined (variable:MC_Segment_75)}
	stMulticarrierModule.i_aifMulticarrierSegments[75]		:= MC_Segment_75;
{END_IF}
{IF defined (variable:MC_Segment_76)}
	stMulticarrierModule.i_aifMulticarrierSegments[76]		:= MC_Segment_76;
{END_IF}
{IF defined (variable:MC_Segment_77)}
 	stMulticarrierModule.i_aifMulticarrierSegments[77]		:= MC_Segment_77;
 {END_IF}
 {IF defined (variable:MC_Segment_78)}
 	stMulticarrierModule.i_aifMulticarrierSegments[78]		:= MC_Segment_78;
 {END_IF}
 {IF defined (variable:MC_Segment_79)}
 	stMulticarrierModule.i_aifMulticarrierSegments[79]		:= MC_Segment_79;
 {END_IF}
  {IF defined (variable:MC_Segment_80)}
 	stMulticarrierModule.i_aifMulticarrierSegments[80]		:= MC_Segment_80;
 {END_IF}
 {IF defined (variable:MC_Segment_81)}
	stMulticarrierModule.i_aifMulticarrierSegments[81]		:= MC_Segment_81;
{END_IF}
{IF defined (variable:MC_Segment_82)}
	stMulticarrierModule.i_aifMulticarrierSegments[82]		:= MC_Segment_82;
{END_IF}
{IF defined (variable:MC_Segment_83)}
	stMulticarrierModule.i_aifMulticarrierSegments[83]		:= MC_Segment_83;
{END_IF}
{IF defined (variable:MC_Segment_84)}
	stMulticarrierModule.i_aifMulticarrierSegments[84]		:= MC_Segment_84;
{END_IF}
{IF defined (variable:MC_Segment_85)}
	stMulticarrierModule.i_aifMulticarrierSegments[85]		:= MC_Segment_85;
{END_IF}
{IF defined (variable:MC_Segment_86)}
	stMulticarrierModule.i_aifMulticarrierSegments[86]		:= MC_Segment_86;
{END_IF}
{IF defined (variable:MC_Segment_87)}
 	stMulticarrierModule.i_aifMulticarrierSegments[87]		:= MC_Segment_87;
 {END_IF}
 {IF defined (variable:MC_Segment_88)}
 	stMulticarrierModule.i_aifMulticarrierSegments[88]		:= MC_Segment_88;
 {END_IF}
 {IF defined (variable:MC_Segment_89)}
 	stMulticarrierModule.i_aifMulticarrierSegments[89]		:= MC_Segment_89;
 {END_IF}
  {IF defined (variable:MC_Segment_90)}
 	stMulticarrierModule.i_aifMulticarrierSegments[90]		:= MC_Segment_90;
 {END_IF}
 {IF defined (variable:MC_Segment_91)}
	stMulticarrierModule.i_aifMulticarrierSegments[91]		:= MC_Segment_91;
{END_IF}
{IF defined (variable:MC_Segment_92)}
	stMulticarrierModule.i_aifMulticarrierSegments[92]		:= MC_Segment_92;
{END_IF}
{IF defined (variable:MC_Segment_93)}
	stMulticarrierModule.i_aifMulticarrierSegments[93]		:= MC_Segment_93;
{END_IF}
{IF defined (variable:MC_Segment_94)}
	stMulticarrierModule.i_aifMulticarrierSegments[94]		:= MC_Segment_94;
{END_IF}
{IF defined (variable:MC_Segment_95)}
	stMulticarrierModule.i_aifMulticarrierSegments[95]		:= MC_Segment_95;
{END_IF}
{IF defined (variable:MC_Segment_96)}
	stMulticarrierModule.i_aifMulticarrierSegments[96]		:= MC_Segment_96;
{END_IF}
{IF defined (variable:MC_Segment_97)}
 	stMulticarrierModule.i_aifMulticarrierSegments[97]		:= MC_Segment_97;
 {END_IF}
 {IF defined (variable:MC_Segment_98)}
 	stMulticarrierModule.i_aifMulticarrierSegments[98]		:= MC_Segment_98;
 {END_IF}
 {IF defined (variable:MC_Segment_99)}
 	stMulticarrierModule.i_aifMulticarrierSegments[99]		:= MC_Segment_99;
 {END_IF}
  {IF defined (variable:MC_Segment_100)}
 	stMulticarrierModule.i_aifMulticarrierSegments[100]		:= MC_Segment_100;
 {END_IF}
END_METHOD

ACTION CheckArraySizeOfTrackElements:
IF GVL_MulticarrierConfiguration.Gc_udiNumberOfCarriers > MCR.GPL.Gc_udiMaxNumberOfCarriers THEN
	xError := TRUE;
	stMachineInterface.q_udiDiagExt	:= ET_DiagExt.InvalidConfiguredParameter;
	stMachineInterface.q_sDiagExt	:= FC_EtDiagExtToString(stMachineInterface.q_udiDiagExt);
	stMachineInterface.q_sMsg := 'Configured Number of Carriers > Number of Carriers in library';
	RETURN;
END_IF

IF GVL_MulticarrierConfiguration.Gc_udiMaxNumberOfSegments > MCR.GPL.Gc_udiMaxNumberOfSegments THEN
	xError := TRUE;
	stMachineInterface.q_udiDiagExt	:= ET_DiagExt.InvalidConfiguredParameter;
	stMachineInterface.q_sDiagExt	:= FC_EtDiagExtToString(stMachineInterface.q_udiDiagExt);
	stMachineInterface.q_sMsg := 'Configured Number of Segments > Number of Segments in library';
	RETURN;
END_IF
END_ACTION

METHOD CreateTrackForSimulation
VAR_INPUT
END_VAR

VAR
	udiIndex: UDINT;
	sTrackConfig: STRING(255);
END_VAR
//--- create String for simulation -------------------------------
FOR udiIndex := 1 TO GVL_MulticarrierConfiguration.Gc_astTracks[1].udiNumberOfSegments DO

	IF GVL_MulticarrierConfiguration.Gc_astSegmentTypes[GVL_MulticarrierConfiguration.Gc_astTracks[1].astSegments[udiIndex].diSegmentTypesIndex].xIsCurved  
	THEN
			sTrackConfig := concat(sTrackConfig ,'C');
	
	ELSE
			sTrackConfig := concat(sTrackConfig,'S');
	
	END_IF

END_FOR

DTC.GVL_OpcUaMulticarrier.G_stMCR.astTracks[1].sGeometry 	:= sTrackConfig;
END_METHOD

METHOD SetCarrierInterfaces
VAR_INPUT
END_VAR
VAR_OUTPUT
	q_xError		: BOOL; 
	q_etDiagExt		: ET_DiagExt;
	q_sResultMsg	: STRING [255];
END_VAR
VAR
	udiIndex: UDINT;
END_VAR
AssignCarriers();

//--- Check if the Array from 1 to NumberCarriers is correctly assigned with Carrier device object
FOR udiIndex := 1 TO GVL_Project.G_udiUsedNumberOfCarriers DO //GVL_MulticarrierConfiguration.Gc_udiNumberOfCarriers DO
	IF stMulticarrierModule.i_aifMulticarrierCarriers[udiIndex] = 0 THEN
		q_xError		:= TRUE;
		q_etDiagExt		:= ET_DiagExt.InvalidConfiguredParameter;
		q_sResultMsg	:= Concat('SetCarrierInterfaces: aifMulticarrierCarrier[',TO_STRING(udiIndex));
		q_sResultMsg	:= Concat(q_sResultMsg,'] = 0');
		RETURN;
	END_IF 
END_FOR

FOR udiIndex := 1 TO MCR.GPL.Gc_udiMaxNumberOfCarriers DO
	
	IF stMulticarrierModule.i_aifMulticarrierCarriers[udiIndex] = 0 THEN
		EXIT;
	END_IF
	
	//--- Set IF_IdentificationMandatory
		xSuccessSetCarrierInterfaces	:= __QUERYINTERFACE(stMulticarrierModule.i_aifMulticarrierCarriers[udiIndex], stMulticarrierModule.i_aifIdentificationMandatory[udiIndex]);
		IF xSuccessSetCarrierInterfaces AND stMulticarrierModule.i_aifIdentificationMandatory[udiIndex] <> 0 THEN
			;
		ELSE
			q_xError		:= TRUE;
			q_etDiagExt		:= ET_DiagExt.InvalidConfiguredParameter;
			q_sResultMsg	:= Concat('SetCarrierInterfaces: aifMulticarrierCarrier[',TO_STRING(udiIndex));
			q_sResultMsg	:= Concat(q_sResultMsg,'] is not supporting IF_IdentificationMandatory');
			RETURN;
		END_IF
		
	//--- Set IF_MovementData
		xSuccessSetCarrierInterfaces	:= __QUERYINTERFACE(stMulticarrierModule.i_aifMulticarrierCarriers[udiIndex], stMulticarrierModule.i_aifMovementDataAccess[udiIndex]);
		IF xSuccessSetCarrierInterfaces AND stMulticarrierModule.i_aifMovementDataAccess[udiIndex] <> 0 THEN
			stMulticarrierModule.i_aifMovementData[udiIndex]	:= stMulticarrierModule.i_aifMovementDataAccess[udiIndex].MovementData;
		ELSE
			q_xError		:= TRUE;
			q_etDiagExt		:= ET_DiagExt.InvalidConfiguredParameter;
			q_sResultMsg	:= Concat('SetCarrierInterfaces: aifMulticarrierCarrier[',TO_STRING(udiIndex));
			q_sResultMsg	:= Concat(q_sResultMsg,'] is not supporting IF_MovementDataAccess');
			RETURN;
		END_IF
		
	//--- Set IF_CarrierState
		xSuccessSetCarrierInterfaces	:= __QUERYINTERFACE(stMulticarrierModule.i_aifMulticarrierCarriers[udiIndex], stMulticarrierModule.i_aifCarrierStateAccess[udiIndex]);
		IF xSuccessSetCarrierInterfaces AND stMulticarrierModule.i_aifCarrierStateAccess[udiIndex] <> 0 THEN
			stMulticarrierModule.i_aifCarrierState[udiIndex]	:= stMulticarrierModule.i_aifCarrierStateAccess[udiIndex].CarrierState;
		ELSE
			q_xError		:= TRUE;
			q_etDiagExt		:= ET_DiagExt.InvalidConfiguredParameter;
			q_sResultMsg	:= Concat('SetCarrierInterfaces: aifMulticarrierCarrier[',TO_STRING(udiIndex));
			q_sResultMsg	:= Concat(q_sResultMsg,'] is not supporting IF_CarrierStateAccess');
			RETURN;
		END_IF
		
	//--- Set IF_CarrierIdentification
		xSuccessSetCarrierInterfaces	:= __QUERYINTERFACE(stMulticarrierModule.i_aifMulticarrierCarriers[udiIndex], stMulticarrierModule.i_aifCarrierIdentificationAccess[udiIndex]);
		IF xSuccessSetCarrierInterfaces AND stMulticarrierModule.i_aifCarrierIdentificationAccess[udiIndex] <> 0 THEN
			stMulticarrierModule.i_aifCarrierIdentification[udiIndex]	:= stMulticarrierModule.i_aifCarrierIdentificationAccess[udiIndex].CarrierIdentification;
		ELSE
			q_xError		:= TRUE;
			q_etDiagExt		:= ET_DiagExt.InvalidConfiguredParameter;
			q_sResultMsg	:= Concat('SetCarrierInterfaces: aifMulticarrierCarrier[',TO_STRING(udiIndex));
			q_sResultMsg	:= Concat(q_sResultMsg,'] is not supporting IF_CarrierIdentificationAccess');
			RETURN;
		END_IF
	
END_FOR

q_xError 		:= FALSE;
q_etDiagExt		:= ET_DiagExt.OK;
q_sResultMsg	:= 'OK';
END_METHOD

METHOD SetCarrierWorkingMode

VAR
	udiIndex: UDINT;
END_VAR
FOR udiIndex := 1 TO MCR.GPL.Gc_udiMaxNumberOfCarriers DO
			
	IF stMulticarrierModule.i_aifCarrierIdentification[udiIndex] <> 0 THEN
		IF udiIndex > GVL_Project.G_udiUsedNumberOfCarriers THEN 
			stMulticarrierModule.i_aifCarrierIdentification[udiIndex].WorkingMode := 2; // 2 = Deactivated
		ELSIF GVL_Project.Gc_xVirtualMulticarrier THEN
			stMulticarrierModule.i_aifCarrierIdentification[udiIndex].WorkingMode := 0; // 0 = Virtual
		ELSE
			stMulticarrierModule.i_aifCarrierIdentification[udiIndex].WorkingMode := 1; // 1 = Real
		END_IF
	ELSE
		;
	END_IF
	
END_FOR
END_METHOD

METHOD SetSegmentInterfaces
VAR_INPUT
END_VAR
VAR_OUTPUT
	q_xError		: BOOL; 
	q_etDiagExt		: ET_DiagExt;
	q_sResultMsg	: STRING [255];
END_VAR
VAR
	udiIndex: UDINT;
END_VAR
AssignSegments();

//--- Check if the Array from 1 to NumberSegments is correctly assigned with Segment device object
FOR udiIndex := 1 TO GVL_MulticarrierConfiguration.Gc_astTracks[1].udiNumberOfSegments DO
	IF stMulticarrierModule.i_aifMulticarrierSegments[udiIndex] = 0 THEN
		q_xError		:= TRUE;
		q_etDiagExt		:= ET_DiagExt.InvalidConfiguredParameter;
		q_sResultMsg	:= Concat('SetSegmentInterfaces: aifMulticarrierSegments[',TO_STRING(udiIndex));
		q_sResultMsg	:= Concat(q_sResultMsg,'] = 0');
		RETURN;
	END_IF 
END_FOR

FOR udiIndex := 1 TO MCR.GPL.Gc_udiMaxNumberOfSegments DO
	 
	IF stMulticarrierModule.i_aifMulticarrierSegments[udiIndex] = 0 THEN
		EXIT;
	END_IF
	
	//--- Set IF_SercosIdentification
		xSuccessSetSegmentInterfaces := __QUERYINTERFACE(stMulticarrierModule.i_aifMulticarrierSegments[udiIndex], stMulticarrierModule.i_aifSegmentSercosIdentificationAccess[udiIndex]);
			
		IF xSuccessSetSegmentInterfaces AND stMulticarrierModule.i_aifSegmentSercosIdentificationAccess[udiIndex] <> 0 THEN
			stMulticarrierModule.i_aifSegmentSercosIdentification[udiIndex]	:= stMulticarrierModule.i_aifSegmentSercosIdentificationAccess[udiIndex].SercosIdentification;
		ELSE
			q_xError		:= TRUE;
			q_etDiagExt		:= ET_DiagExt.InvalidConfiguredParameter;
			q_sResultMsg	:= Concat('SetSegmentInterfaces: MulticarrierSegment[',TO_STRING(udiIndex));
			q_sResultMsg	:= Concat(q_sResultMsg,'] is not supporting IF_SercosIdentificationAccess');
			RETURN;
		END_IF
	
	//--- Set IF_SegmentEnable
		xSuccessSetSegmentInterfaces := __QUERYINTERFACE(stMulticarrierModule.i_aifMulticarrierSegments[udiIndex], stMulticarrierModule.i_aifSegmentEnableAccess[udiIndex]);
			
		IF xSuccessSetSegmentInterfaces AND stMulticarrierModule.i_aifSegmentEnableAccess[udiIndex] <> 0 THEN
			stMulticarrierModule.i_aifSegmentEnable[udiIndex]	:= stMulticarrierModule.i_aifSegmentEnableAccess[udiIndex].SegmentEnable;
		ELSE
			q_xError		:= TRUE;
			q_etDiagExt		:= ET_DiagExt.InvalidConfiguredParameter;
			q_sResultMsg	:= Concat('SetSegmentInterfaces: MulticarrierSegment[',TO_STRING(udiIndex));
			q_sResultMsg	:= Concat(q_sResultMsg,'] is not supporting IF_SegmentEnableAccess');
			RETURN;
		END_IF
		
	//--- Set IF_SegmentGeometry
		xSuccessSetSegmentInterfaces := __QUERYINTERFACE(stMulticarrierModule.i_aifMulticarrierSegments[udiIndex], stMulticarrierModule.i_aifSegmentGeometryAccess[udiIndex]);
			
		IF xSuccessSetSegmentInterfaces AND stMulticarrierModule.i_aifSegmentGeometryAccess[udiIndex] <> 0 THEN
			stMulticarrierModule.i_aifSegmentGeometry[udiIndex]	:= stMulticarrierModule.i_aifSegmentGeometryAccess[udiIndex].SegmentGeometry;
		ELSE
			q_xError		:= TRUE;
			q_etDiagExt		:= ET_DiagExt.InvalidConfiguredParameter;
			q_sResultMsg	:= Concat('SetSegmentInterfaces: MulticarrierSegment[',TO_STRING(udiIndex));
			q_sResultMsg	:= Concat(q_sResultMsg,'] is not supporting IF_SegmentGeometryAccess');
			RETURN;
		END_IF
END_FOR


q_xError 		:= FALSE;
q_etDiagExt		:= ET_DiagExt.OK;
q_sResultMsg	:= 'OK';
END_METHOD

METHOD SetSegmentWorkingMode


VAR
	udiIndex: UDINT;
END_VAR
FOR udiIndex := 1 TO MCR.GPL.Gc_udiMaxNumberOfSegments DO
			
	IF stMulticarrierModule.i_aifSegmentSercosIdentification[udiIndex] <> 0 THEN
		IF udiIndex > GVL_MulticarrierConfiguration.Gc_astTracks[1].udiNumberOfSegments THEN
			stMulticarrierModule.i_aifSegmentSercosIdentification[udiIndex].WorkingMode := 2; // 2 = Deactivated
		ELSIF GVL_Project.Gc_xVirtualMulticarrier THEN
			stMulticarrierModule.i_aifSegmentSercosIdentification[udiIndex].WorkingMode := 0; // 0 = Virtual
		ELSE
			stMulticarrierModule.i_aifSegmentSercosIdentification[udiIndex].WorkingMode := 1; // 1 = Real
		END_IF
	ELSE
		;
	END_IF
END_FOR
END_METHOD

METHOD SetTrackInterfaces
VAR_INPUT
END_VAR
VAR_OUTPUT
	q_xError		: BOOL; 
	q_etDiagExt		: ET_DiagExt;
	q_sResultMsg	: STRING [255];
END_VAR
VAR
	udiIndex: UDINT;
	
END_VAR
//--- Assign the Track here.
	stMulticarrierModule.i_ifMulticarrierTrack		:= MC_Track_1;
  
//--- Check if the Array from 1 to NumberSegments is correctly assigned with Segment device object
IF stMulticarrierModule.i_ifMulticarrierTrack = 0 THEN
		q_xError		:= TRUE;
		q_etDiagExt		:= ET_DiagExt.InvalidConfiguredParameter;
		q_sResultMsg	:= 'SetTrackInterfaces: i_ifMulticarrierTrack = 0';
		RETURN;
	END_IF 


//--- Set IF_TrackEnable
	xSuccessSetTrackInterfaces := __QUERYINTERFACE(stMulticarrierModule.i_ifMulticarrierTrack, stMulticarrierModule.i_ifMulticarrierTrackEnableAccess);
		
	IF xSuccessSetTrackInterfaces AND stMulticarrierModule.i_ifMulticarrierTrackEnableAccess <> 0 THEN
		stMulticarrierModule.i_ifMulticarrierTrackEnable	:= stMulticarrierModule.i_ifMulticarrierTrackEnableAccess.TrackEnable;
	ELSE
		q_xError		:= TRUE;
		q_etDiagExt		:= ET_DiagExt.InvalidConfiguredParameter;
		q_sResultMsg	:= 'SetTrackInterfaces: MulticarrierTrack is not supporting IF_TrackEnableAccess';
		RETURN;
	END_IF

q_xError 		:= FALSE;
q_etDiagExt		:= ET_DiagExt.OK;
q_sResultMsg	:= 'OK';
END_METHOD

METHOD WriteGeometryOnSegments
VAR_INPUT
END_VAR

VAR
	udiIndex: UDINT;
	iResidualValue: INT;
END_VAR
FOR udiIndex := 1 TO GVL_MulticarrierConfiguration.Gc_astTracks[1].udiNumberOfSegments DO
		
		//-- set length
		stMulticarrierModule.i_aifSegmentGeometry[udiIndex].ConfiguredLength 
					:= GVL_MulticarrierConfiguration.Gc_astSegmentTypes[GVL_MulticarrierConfiguration.Gc_astTracks[1].astSegments[udiIndex].diSegmentTypesIndex].lrRailLength;
		
		//-- set Denominator
		stMulticarrierModule.i_aifSegmentGeometry[udiIndex].ConfiguredAngleFractionDenominator 
					:= GVL_MulticarrierConfiguration.Gc_astSegmentTypes[GVL_MulticarrierConfiguration.Gc_astTracks[1].astSegments[udiIndex].diSegmentTypesIndex].udiAngleFractionDenominator;
					
		//-- set Numerator
		stMulticarrierModule.i_aifSegmentGeometry[udiIndex].ConfiguredAngleFractionNumerator   
					:= GVL_MulticarrierConfiguration.Gc_astSegmentTypes[GVL_MulticarrierConfiguration.Gc_astTracks[1].astSegments[udiIndex].diSegmentTypesIndex].diAngleFractionNumerator;
			
	END_FOR
END_METHOD

ACTION _aBrakeReleaseStep_active:
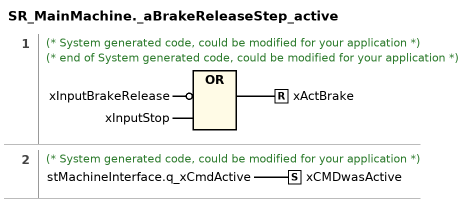
// NETWORK 1
// 					(* System generated code, could be modified for your application *)
// (* end of System generated code, could be modified for your application *)
//
xActBrake R= NOT xInputBrakeRelease OR xInputStop;

// NETWORK 2
// (* System generated code, could be modified for your application *)
xCMDwasActive S= stMachineInterface.q_xCmdActive;
END_ACTION

ACTION _aBrakeReleaseStep_entry:
(* System generated code, could be modified for your application *)
	xCMDwasActive		:= FALSE;
	stMachineInterface.iq_diCmd	:= ET_Cmd.BrakeRelease;
(* End of system generated code, could be modified for your application *)
END_ACTION

ACTION AutoStep_Action:
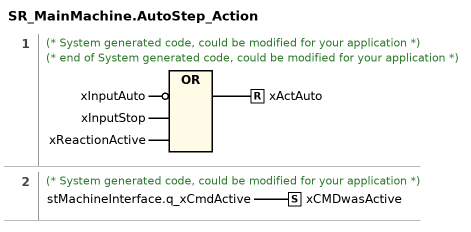
// NETWORK 1
// 					(* System generated code, could be modified for your application *)
// (* end of System generated code, could be modified for your application *)
//
xActAuto R= NOT xInputAuto OR xInputStop OR xReactionActive;

// NETWORK 2
// (* System generated code, could be modified for your application *)
xCMDwasActive S= stMachineInterface.q_xCmdActive;
END_ACTION

ACTION AutoStep_Entry:
(* System generated code, could be modified for your application *)
	xCmdWasActive := FALSE;
	stMachineInterface.iq_diCmd := ET_Cmd.Auto;
(* End of system generated code, could be modified for your application *)
END_ACTION

ACTION AutoStop_Action:
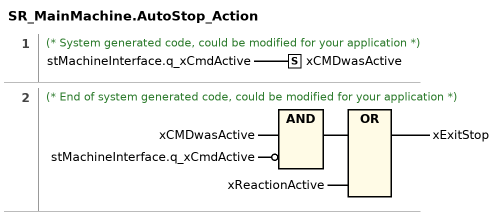
// NETWORK 1
// (* System generated code, could be modified for your application *)
xCMDwasActive S= stMachineInterface.q_xCmdActive;

